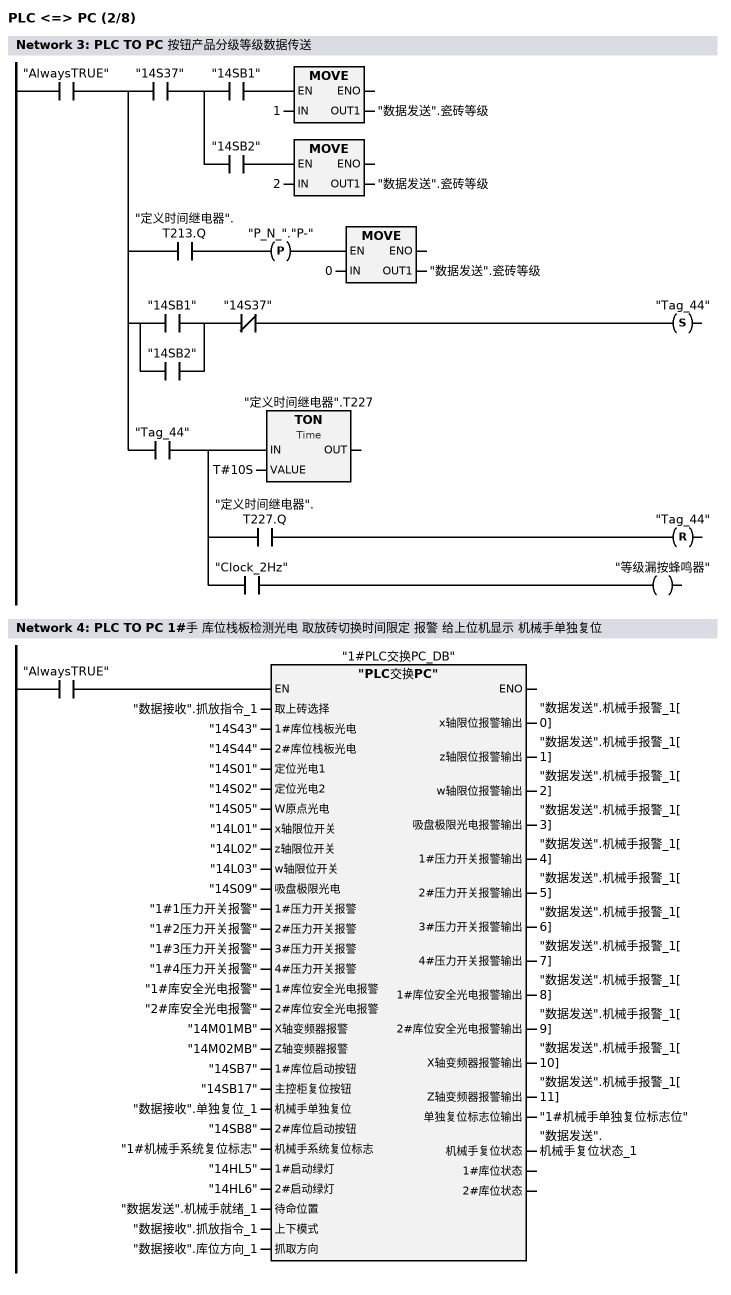
   #_w1 := "AlwaysTRUE" AND "14S37";
   IF #_w1 AND "14SB1" THEN "数据发送".瓷砖等级 := 1; END_IF;
   IF #_w1 AND "14SB2" THEN "数据发送".瓷砖等级 := 2; END_IF;
   #_w2 := "AlwaysTRUE" AND "定义时间继电器".T213.Q;
   #_w3 := #_w2 AND NOT "P_N_"."P-";   // rising edge
   "P_N_"."P-" := #_w2;
   IF #_w3 THEN "数据发送".瓷砖等级 := 0; END_IF;
   IF "AlwaysTRUE" AND ("14SB1" OR "14SB2") AND NOT "14S37" THEN "Tag_44" := TRUE; END_IF;
   #_w4 := "AlwaysTRUE" AND "Tag_44";
   "定义时间继电器".T227.TON(IN := #_w4, PT := T#10S);   // TON coil
   IF #_w4 AND "定义时间继电器".T227.Q THEN "Tag_44" := FALSE; END_IF;
   "等级漏按蜂鸣器" := #_w4 AND "Clock_2Hz";
END_REGION

REGION Network 4: PLC TO PC 1#手 库位栈板检测光电 取放砖切换时间限定 报警 给上位机显示 机械手单独复位
   RUNG wire#powerrail
      Contact( "AlwaysTRUE" )
      "1#PLC交换PC_DB"(取上砖选择 := "数据接收".抓放指令_1, "1#库位栈板光电" := "14S43", "2#库位栈板光电" := "14S44", 定位光电1 := "14S01", 定位光电2 := "14S02", W原点光电 := "14S05", x轴限位开关 := "14L01", z轴限位开关 := "14L02", w轴限位开关 := "14L03", 吸盘极限光电 := "14S09", "1#压力开关报警" := "1#1压力开关报警", "2#压力开关报警" := "1#2压力开关报警", "3#压力开关报警" := "1#3压力开关报警", "4#压力开关报警" := "1#4压力开关报警", "1#库位安全光电报警" := "1#库安全光电报警", "2#库位安全光电报警" := "2#库安全光电报警", X轴变频器报警 := "14M01MB", Z轴变频器报警 := "14M02MB", "1#库位启动按钮" := "14SB7", 主控柜复位按钮 := "14SB17", 机械手单独复位 := "数据接收".单独复位_1, "2#库位启动按钮" := "14SB8", 机械手系统复位标志 := "1#机械手系统复位标志", "1#启动绿灯" := "14HL5", "2#启动绿灯" := "14HL6", 待命位置 := "数据发送".机械手就绪_1, 上下模式 := "数据接收".抓放指令_1, 抓取方向 := "数据接收".库位方向_1, x轴限位报警输出 => "数据发送".机械手报警_1[0], z轴限位报警输出 => "数据发送".机械手报警_1[1], w轴限位报警输出 => "数据发送".机械手报警_1[2], 吸盘极限光电报警输出 => "数据发送".机械手报警_1[3], "1#压力开关报警输出" => "数据发送".机械手报警_1[4], "2#压力开关报警输出" => "数据发送".机械手报警_1[5], "3#压力开关报警输出" => "数据发送".机械手报警_1[6], "4#压力开关报警输出" => "数据发送".机械手报警_1[7], "1#库位安全光电报警输出" => "数据发送".机械手报警_1[8], "2#库位安全光电报警输出" => "数据发送".机械手报警_1[9], X轴变频器报警输出 => "数据发送".机械手报警_1[10], Z轴变频器报警输出 => "数据发送".机械手报警_1[11], 单独复位标志位输出 => "1#机械手单独复位标志位", 机械手复位状态 => "数据发送".机械手复位状态_1, "1#库位状态" =>, "2#库位状态" =>)
   END_RUNG
   // the same network as SCL:
   IF "AlwaysTRUE" THEN
       "1#PLC交换PC_DB"(取上砖选择 := "数据接收".抓放指令_1,   // "PLC交换PC"
                      "1#库位栈板光电" := "14S43",
                      "2#库位栈板光电" := "14S44",
                      定位光电1 := "14S01",
                      定位光电2 := "14S02",
                      W原点光电 := "14S05",
                      x轴限位开关 := "14L01",
                      z轴限位开关 := "14L02",
                      w轴限位开关 := "14L03",
                      吸盘极限光电 := "14S09",
                      "1#压力开关报警" := "1#1压力开关报警",
                      "2#压力开关报警" := "1#2压力开关报警",
                      "3#压力开关报警" := "1#3压力开关报警",
                      "4#压力开关报警" := "1#4压力开关报警",
                      "1#库位安全光电报警" := "1#库安全光电报警",
                      "2#库位安全光电报警" := "2#库安全光电报警",
                      X轴变频器报警 := "14M01MB",
                      Z轴变频器报警 := "14M02MB",
                      "1#库位启动按钮" := "14SB7",
                      主控柜复位按钮 := "14SB17",
                      机械手单独复位 := "数据接收".单独复位_1,
                      "2#库位启动按钮" := "14SB8",
                      机械手系统复位标志 := "1#机械手系统复位标志",
                      "1#启动绿灯" := "14HL5",
                      "2#启动绿灯" := "14HL6",
                      待命位置 := "数据发送".机械手就绪_1,
                      上下模式 := "数据接收".抓放指令_1,
                      抓取方向 := "数据接收".库位方向_1,
                      x轴限位报警输出 => "数据发送".机械手报警_1[0],
                      z轴限位报警输出 => "数据发送".机械手报警_1[1],
                      w轴限位报警输出 => "数据发送".机械手报警_1[2],
                      吸盘极限光电报警输出 => "数据发送".机械手报警_1[3],
                      "1#压力开关报警输出" => "数据发送".机械手报警_1[4],
                      "2#压力开关报警输出" => "数据发送".机械手报警_1[5],
                      "3#压力开关报警输出" => "数据发送".机械手报警_1[6],
                      "4#压力开关报警输出" => "数据发送".机械手报警_1[7],
                      "1#库位安全光电报警输出" => "数据发送".机械手报警_1[8],
                      "2#库位安全光电报警输出" => "数据发送".机械手报警_1[9],
                      X轴变频器报警输出 => "数据发送".机械手报警_1[10],
                      Z轴变频器报警输出 => "数据发送".机械手报警_1[11],
                      单独复位标志位输出 => "1#机械手单独复位标志位",
                      机械手复位状态 => "数据发送".机械手复位状态_1);
   END_IF;
END_REGION

REGION Network 5: PLC TO PC 2#手 库位栈板检测光电 取放砖切换时间限定 报警 给上位机显示 机械手单独复位
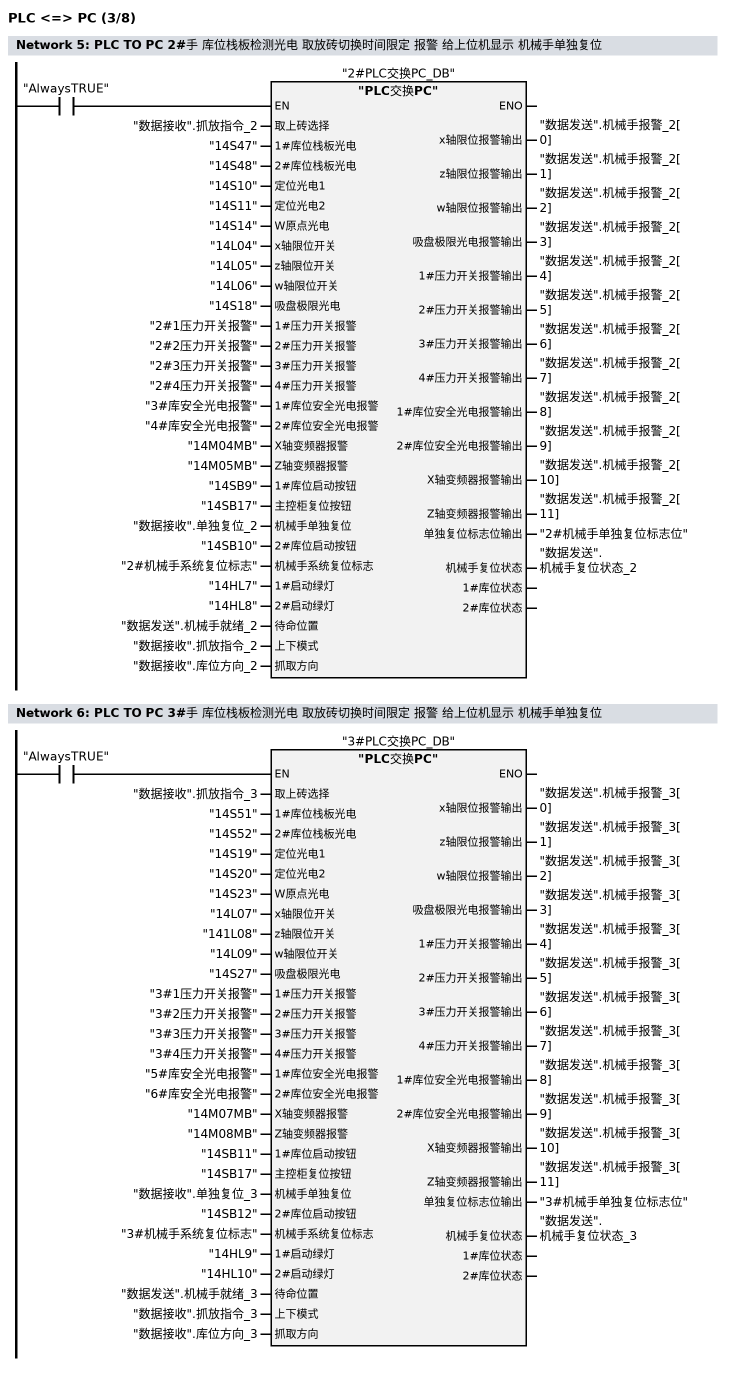
   RUNG wire#powerrail
      Contact( "AlwaysTRUE" )
      "2#PLC交换PC_DB"(取上砖选择 := "数据接收".抓放指令_2, "1#库位栈板光电" := "14S47", "2#库位栈板光电" := "14S48", 定位光电1 := "14S10", 定位光电2 := "14S11", W原点光电 := "14S14", x轴限位开关 := "14L04", z轴限位开关 := "14L05", w轴限位开关 := "14L06", 吸盘极限光电 := "14S18", "1#压力开关报警" := "2#1压力开关报警", "2#压力开关报警" := "2#2压力开关报警", "3#压力开关报警" := "2#3压力开关报警", "4#压力开关报警" := "2#4压力开关报警", "1#库位安全光电报警" := "3#库安全光电报警", "2#库位安全光电报警" := "4#库安全光电报警", X轴变频器报警 := "14M04MB", Z轴变频器报警 := "14M05MB", "1#库位启动按钮" := "14SB9", 主控柜复位按钮 := "14SB17", 机械手单独复位 := "数据接收".单独复位_2, "2#库位启动按钮" := "14SB10", 机械手系统复位标志 := "2#机械手系统复位标志", "1#启动绿灯" := "14HL7", "2#启动绿灯" := "14HL8", 待命位置 := "数据发送".机械手就绪_2, 上下模式 := "数据接收".抓放指令_2, 抓取方向 := "数据接收".库位方向_2, x轴限位报警输出 => "数据发送".机械手报警_2[0], z轴限位报警输出 => "数据发送".机械手报警_2[1], w轴限位报警输出 => "数据发送".机械手报警_2[2], 吸盘极限光电报警输出 => "数据发送".机械手报警_2[3], "1#压力开关报警输出" => "数据发送".机械手报警_2[4], "2#压力开关报警输出" => "数据发送".机械手报警_2[5], "3#压力开关报警输出" => "数据发送".机械手报警_2[6], "4#压力开关报警输出" => "数据发送".机械手报警_2[7], "1#库位安全光电报警输出" => "数据发送".机械手报警_2[8], "2#库位安全光电报警输出" => "数据发送".机械手报警_2[9], X轴变频器报警输出 => "数据发送".机械手报警_2[10], Z轴变频器报警输出 => "数据发送".机械手报警_2[11], 单独复位标志位输出 => "2#机械手单独复位标志位", 机械手复位状态 => "数据发送".机械手复位状态_2, "1#库位状态" =>, "2#库位状态" =>)
   END_RUNG
   // the same network as SCL:
   IF "AlwaysTRUE" THEN
       "2#PLC交换PC_DB"(取上砖选择 := "数据接收".抓放指令_2,   // "PLC交换PC"
                      "1#库位栈板光电" := "14S47",
                      "2#库位栈板光电" := "14S48",
                      定位光电1 := "14S10",
                      定位光电2 := "14S11",
                      W原点光电 := "14S14",
                      x轴限位开关 := "14L04",
                      z轴限位开关 := "14L05",
                      w轴限位开关 := "14L06",
                      吸盘极限光电 := "14S18",
                      "1#压力开关报警" := "2#1压力开关报警",
                      "2#压力开关报警" := "2#2压力开关报警",
                      "3#压力开关报警" := "2#3压力开关报警",
                      "4#压力开关报警" := "2#4压力开关报警",
                      "1#库位安全光电报警" := "3#库安全光电报警",
                      "2#库位安全光电报警" := "4#库安全光电报警",
                      X轴变频器报警 := "14M04MB",
                      Z轴变频器报警 := "14M05MB",
                      "1#库位启动按钮" := "14SB9",
                      主控柜复位按钮 := "14SB17",
                      机械手单独复位 := "数据接收".单独复位_2,
                      "2#库位启动按钮" := "14SB10",
                      机械手系统复位标志 := "2#机械手系统复位标志",
                      "1#启动绿灯" := "14HL7",
                      "2#启动绿灯" := "14HL8",
                      待命位置 := "数据发送".机械手就绪_2,
                      上下模式 := "数据接收".抓放指令_2,
                      抓取方向 := "数据接收".库位方向_2,
                      x轴限位报警输出 => "数据发送".机械手报警_2[0],
                      z轴限位报警输出 => "数据发送".机械手报警_2[1],
                      w轴限位报警输出 => "数据发送".机械手报警_2[2],
                      吸盘极限光电报警输出 => "数据发送".机械手报警_2[3],
                      "1#压力开关报警输出" => "数据发送".机械手报警_2[4],
                      "2#压力开关报警输出" => "数据发送".机械手报警_2[5],
                      "3#压力开关报警输出" => "数据发送".机械手报警_2[6],
                      "4#压力开关报警输出" => "数据发送".机械手报警_2[7],
                      "1#库位安全光电报警输出" => "数据发送".机械手报警_2[8],
                      "2#库位安全光电报警输出" => "数据发送".机械手报警_2[9],
                      X轴变频器报警输出 => "数据发送".机械手报警_2[10],
                      Z轴变频器报警输出 => "数据发送".机械手报警_2[11],
                      单独复位标志位输出 => "2#机械手单独复位标志位",
                      机械手复位状态 => "数据发送".机械手复位状态_2);
   END_IF;
END_REGION

REGION Network 6: PLC TO PC 3#手 库位栈板检测光电 取放砖切换时间限定 报警 给上位机显示 机械手单独复位
   RUNG wire#powerrail
      Contact( "AlwaysTRUE" )
      "3#PLC交换PC_DB"(取上砖选择 := "数据接收".抓放指令_3, "1#库位栈板光电" := "14S51", "2#库位栈板光电" := "14S52", 定位光电1 := "14S19", 定位光电2 := "14S20", W原点光电 := "14S23", x轴限位开关 := "14L07", z轴限位开关 := "141L08", w轴限位开关 := "14L09", 吸盘极限光电 := "14S27", "1#压力开关报警" := "3#1压力开关报警", "2#压力开关报警" := "3#2压力开关报警", "3#压力开关报警" := "3#3压力开关报警", "4#压力开关报警" := "3#4压力开关报警", "1#库位安全光电报警" := "5#库安全光电报警", "2#库位安全光电报警" := "6#库安全光电报警", X轴变频器报警 := "14M07MB", Z轴变频器报警 := "14M08MB", "1#库位启动按钮" := "14SB11", 主控柜复位按钮 := "14SB17", 机械手单独复位 := "数据接收".单独复位_3, "2#库位启动按钮" := "14SB12", 机械手系统复位标志 := "3#机械手系统复位标志", "1#启动绿灯" := "14HL9", "2#启动绿灯" := "14HL10", 待命位置 := "数据发送".机械手就绪_3, 上下模式 := "数据接收".抓放指令_3, 抓取方向 := "数据接收".库位方向_3, x轴限位报警输出 => "数据发送".机械手报警_3[0], z轴限位报警输出 => "数据发送".机械手报警_3[1], w轴限位报警输出 => "数据发送".机械手报警_3[2], 吸盘极限光电报警输出 => "数据发送".机械手报警_3[3], "1#压力开关报警输出" => "数据发送".机械手报警_3[4], "2#压力开关报警输出" => "数据发送".机械手报警_3[5], "3#压力开关报警输出" => "数据发送".机械手报警_3[6], "4#压力开关报警输出" => "数据发送".机械手报警_3[7], "1#库位安全光电报警输出" => "数据发送".机械手报警_3[8], "2#库位安全光电报警输出" => "数据发送".机械手报警_3[9], X轴变频器报警输出 => "数据发送".机械手报警_3[10], Z轴变频器报警输出 => "数据发送".机械手报警_3[11], 单独复位标志位输出 => "3#机械手单独复位标志位", 机械手复位状态 => "数据发送".机械手复位状态_3, "1#库位状态" =>, "2#库位状态" =>)
   END_RUNG
   // the same network as SCL:
   IF "AlwaysTRUE" THEN
       "3#PLC交换PC_DB"(取上砖选择 := "数据接收".抓放指令_3,   // "PLC交换PC"
                      "1#库位栈板光电" := "14S51",
                      "2#库位栈板光电" := "14S52",
                      定位光电1 := "14S19",
                      定位光电2 := "14S20",
                      W原点光电 := "14S23",
                      x轴限位开关 := "14L07",
                      z轴限位开关 := "141L08",
                      w轴限位开关 := "14L09",
                      吸盘极限光电 := "14S27",
                      "1#压力开关报警" := "3#1压力开关报警",
                      "2#压力开关报警" := "3#2压力开关报警",
                      "3#压力开关报警" := "3#3压力开关报警",
                      "4#压力开关报警" := "3#4压力开关报警",
                      "1#库位安全光电报警" := "5#库安全光电报警",
                      "2#库位安全光电报警" := "6#库安全光电报警",
                      X轴变频器报警 := "14M07MB",
                      Z轴变频器报警 := "14M08MB",
                      "1#库位启动按钮" := "14SB11",
                      主控柜复位按钮 := "14SB17",
                      机械手单独复位 := "数据接收".单独复位_3,
                      "2#库位启动按钮" := "14SB12",
                      机械手系统复位标志 := "3#机械手系统复位标志",
                      "1#启动绿灯" := "14HL9",
                      "2#启动绿灯" := "14HL10",
                      待命位置 := "数据发送".机械手就绪_3,
                      上下模式 := "数据接收".抓放指令_3,
                      抓取方向 := "数据接收".库位方向_3,
                      x轴限位报警输出 => "数据发送".机械手报警_3[0],
                      z轴限位报警输出 => "数据发送".机械手报警_3[1],
                      w轴限位报警输出 => "数据发送".机械手报警_3[2],
                      吸盘极限光电报警输出 => "数据发送".机械手报警_3[3],
                      "1#压力开关报警输出" => "数据发送".机械手报警_3[4],
                      "2#压力开关报警输出" => "数据发送".机械手报警_3[5],
                      "3#压力开关报警输出" => "数据发送".机械手报警_3[6],
                      "4#压力开关报警输出" => "数据发送".机械手报警_3[7],
                      "1#库位安全光电报警输出" => "数据发送".机械手报警_3[8],
                      "2#库位安全光电报警输出" => "数据发送".机械手报警_3[9],
                      X轴变频器报警输出 => "数据发送".机械手报警_3[10],
                      Z轴变频器报警输出 => "数据发送".机械手报警_3[11],
                      单独复位标志位输出 => "3#机械手单独复位标志位",
                      机械手复位状态 => "数据发送".机械手复位状态_3);
   END_IF;
END_REGION

REGION Network 7: PLC TO PC 4#手 库位栈板检测光电 取放砖切换时间限定 报警 给上位机显示 机械手单独复位
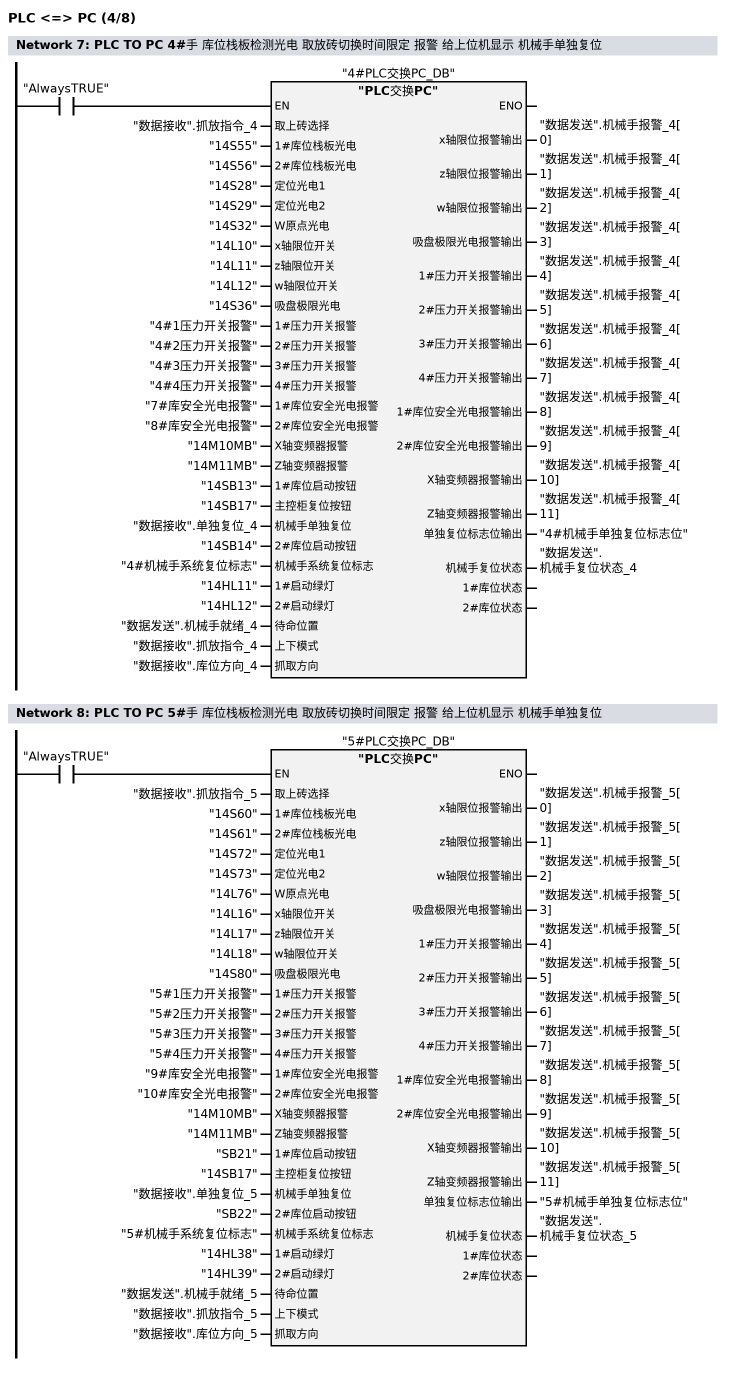
   RUNG wire#powerrail
      Contact( "AlwaysTRUE" )
      "4#PLC交换PC_DB"(取上砖选择 := "数据接收".抓放指令_4, "1#库位栈板光电" := "14S55", "2#库位栈板光电" := "14S56", 定位光电1 := "14S28", 定位光电2 := "14S29", W原点光电 := "14S32", x轴限位开关 := "14L10", z轴限位开关 := "14L11", w轴限位开关 := "14L12", 吸盘极限光电 := "14S36", "1#压力开关报警" := "4#1压力开关报警", "2#压力开关报警" := "4#2压力开关报警", "3#压力开关报警" := "4#3压力开关报警", "4#压力开关报警" := "4#4压力开关报警", "1#库位安全光电报警" := "7#库安全光电报警", "2#库位安全光电报警" := "8#库安全光电报警", X轴变频器报警 := "14M10MB", Z轴变频器报警 := "14M11MB", "1#库位启动按钮" := "14SB13", 主控柜复位按钮 := "14SB17", 机械手单独复位 := "数据接收".单独复位_4, "2#库位启动按钮" := "14SB14", 机械手系统复位标志 := "4#机械手系统复位标志", "1#启动绿灯" := "14HL11", "2#启动绿灯" := "14HL12", 待命位置 := "数据发送".机械手就绪_4, 上下模式 := "数据接收".抓放指令_4, 抓取方向 := "数据接收".库位方向_4, x轴限位报警输出 => "数据发送".机械手报警_4[0], z轴限位报警输出 => "数据发送".机械手报警_4[1], w轴限位报警输出 => "数据发送".机械手报警_4[2], 吸盘极限光电报警输出 => "数据发送".机械手报警_4[3], "1#压力开关报警输出" => "数据发送".机械手报警_4[4], "2#压力开关报警输出" => "数据发送".机械手报警_4[5], "3#压力开关报警输出" => "数据发送".机械手报警_4[6], "4#压力开关报警输出" => "数据发送".机械手报警_4[7], "1#库位安全光电报警输出" => "数据发送".机械手报警_4[8], "2#库位安全光电报警输出" => "数据发送".机械手报警_4[9], X轴变频器报警输出 => "数据发送".机械手报警_4[10], Z轴变频器报警输出 => "数据发送".机械手报警_4[11], 单独复位标志位输出 => "4#机械手单独复位标志位", 机械手复位状态 => "数据发送".机械手复位状态_4, "1#库位状态" =>, "2#库位状态" =>)
   END_RUNG
   // the same network as SCL:
   IF "AlwaysTRUE" THEN
       "4#PLC交换PC_DB"(取上砖选择 := "数据接收".抓放指令_4,   // "PLC交换PC"
                      "1#库位栈板光电" := "14S55",
                      "2#库位栈板光电" := "14S56",
                      定位光电1 := "14S28",
                      定位光电2 := "14S29",
                      W原点光电 := "14S32",
                      x轴限位开关 := "14L10",
                      z轴限位开关 := "14L11",
                      w轴限位开关 := "14L12",
                      吸盘极限光电 := "14S36",
                      "1#压力开关报警" := "4#1压力开关报警",
                      "2#压力开关报警" := "4#2压力开关报警",
                      "3#压力开关报警" := "4#3压力开关报警",
                      "4#压力开关报警" := "4#4压力开关报警",
                      "1#库位安全光电报警" := "7#库安全光电报警",
                      "2#库位安全光电报警" := "8#库安全光电报警",
                      X轴变频器报警 := "14M10MB",
                      Z轴变频器报警 := "14M11MB",
                      "1#库位启动按钮" := "14SB13",
                      主控柜复位按钮 := "14SB17",
                      机械手单独复位 := "数据接收".单独复位_4,
                      "2#库位启动按钮" := "14SB14",
                      机械手系统复位标志 := "4#机械手系统复位标志",
                      "1#启动绿灯" := "14HL11",
                      "2#启动绿灯" := "14HL12",
                      待命位置 := "数据发送".机械手就绪_4,
                      上下模式 := "数据接收".抓放指令_4,
                      抓取方向 := "数据接收".库位方向_4,
                      x轴限位报警输出 => "数据发送".机械手报警_4[0],
                      z轴限位报警输出 => "数据发送".机械手报警_4[1],
                      w轴限位报警输出 => "数据发送".机械手报警_4[2],
                      吸盘极限光电报警输出 => "数据发送".机械手报警_4[3],
                      "1#压力开关报警输出" => "数据发送".机械手报警_4[4],
                      "2#压力开关报警输出" => "数据发送".机械手报警_4[5],
                      "3#压力开关报警输出" => "数据发送".机械手报警_4[6],
                      "4#压力开关报警输出" => "数据发送".机械手报警_4[7],
                      "1#库位安全光电报警输出" => "数据发送".机械手报警_4[8],
                      "2#库位安全光电报警输出" => "数据发送".机械手报警_4[9],
                      X轴变频器报警输出 => "数据发送".机械手报警_4[10],
                      Z轴变频器报警输出 => "数据发送".机械手报警_4[11],
                      单独复位标志位输出 => "4#机械手单独复位标志位",
                      机械手复位状态 => "数据发送".机械手复位状态_4);
   END_IF;
END_REGION

REGION Network 8: PLC TO PC 5#手 库位栈板检测光电 取放砖切换时间限定 报警 给上位机显示 机械手单独复位
   RUNG wire#powerrail
      Contact( "AlwaysTRUE" )
      "5#PLC交换PC_DB"(取上砖选择 := "数据接收".抓放指令_5, "1#库位栈板光电" := "14S60", "2#库位栈板光电" := "14S61", 定位光电1 := "14S72", 定位光电2 := "14S73", W原点光电 := "14L76", x轴限位开关 := "14L16", z轴限位开关 := "14L17", w轴限位开关 := "14L18", 吸盘极限光电 := "14S80", "1#压力开关报警" := "5#1压力开关报警", "2#压力开关报警" := "5#2压力开关报警", "3#压力开关报警" := "5#3压力开关报警", "4#压力开关报警" := "5#4压力开关报警", "1#库位安全光电报警" := "9#库安全光电报警", "2#库位安全光电报警" := "10#库安全光电报警", X轴变频器报警 := "14M10MB", Z轴变频器报警 := "14M11MB", "1#库位启动按钮" := "SB21", 主控柜复位按钮 := "14SB17", 机械手单独复位 := "数据接收".单独复位_5, "2#库位启动按钮" := "SB22", 机械手系统复位标志 := "5#机械手系统复位标志", "1#启动绿灯" := "14HL38", "2#启动绿灯" := "14HL39", 待命位置 := "数据发送".机械手就绪_5, 上下模式 := "数据接收".抓放指令_5, 抓取方向 := "数据接收".库位方向_5, x轴限位报警输出 => "数据发送".机械手报警_5[0], z轴限位报警输出 => "数据发送".机械手报警_5[1], w轴限位报警输出 => "数据发送".机械手报警_5[2], 吸盘极限光电报警输出 => "数据发送".机械手报警_5[3], "1#压力开关报警输出" => "数据发送".机械手报警_5[4], "2#压力开关报警输出" => "数据发送".机械手报警_5[5], "3#压力开关报警输出" => "数据发送".机械手报警_5[6], "4#压力开关报警输出" => "数据发送".机械手报警_5[7], "1#库位安全光电报警输出" => "数据发送".机械手报警_5[8], "2#库位安全光电报警输出" => "数据发送".机械手报警_5[9], X轴变频器报警输出 => "数据发送".机械手报警_5[10], Z轴变频器报警输出 => "数据发送".机械手报警_5[11], 单独复位标志位输出 => "5#机械手单独复位标志位", 机械手复位状态 => "数据发送".机械手复位状态_5, "1#库位状态" =>, "2#库位状态" =>)
   END_RUNG
   // the same network as SCL:
   IF "AlwaysTRUE" THEN
       "5#PLC交换PC_DB"(取上砖选择 := "数据接收".抓放指令_5,   // "PLC交换PC"
                      "1#库位栈板光电" := "14S60",
                      "2#库位栈板光电" := "14S61",
                      定位光电1 := "14S72",
                      定位光电2 := "14S73",
                      W原点光电 := "14L76",
                      x轴限位开关 := "14L16",
                      z轴限位开关 := "14L17",
                      w轴限位开关 := "14L18",
                      吸盘极限光电 := "14S80",
                      "1#压力开关报警" := "5#1压力开关报警",
                      "2#压力开关报警" := "5#2压力开关报警",
                      "3#压力开关报警" := "5#3压力开关报警",
                      "4#压力开关报警" := "5#4压力开关报警",
                      "1#库位安全光电报警" := "9#库安全光电报警",
                      "2#库位安全光电报警" := "10#库安全光电报警",
                      X轴变频器报警 := "14M10MB",
                      Z轴变频器报警 := "14M11MB",
                      "1#库位启动按钮" := "SB21",
                      主控柜复位按钮 := "14SB17",
                      机械手单独复位 := "数据接收".单独复位_5,
                      "2#库位启动按钮" := "SB22",
                      机械手系统复位标志 := "5#机械手系统复位标志",
                      "1#启动绿灯" := "14HL38",
                      "2#启动绿灯" := "14HL39",
                      待命位置 := "数据发送".机械手就绪_5,
                      上下模式 := "数据接收".抓放指令_5,
                      抓取方向 := "数据接收".库位方向_5,
                      x轴限位报警输出 => "数据发送".机械手报警_5[0],
                      z轴限位报警输出 => "数据发送".机械手报警_5[1],
                      w轴限位报警输出 => "数据发送".机械手报警_5[2],
                      吸盘极限光电报警输出 => "数据发送".机械手报警_5[3],
                      "1#压力开关报警输出" => "数据发送".机械手报警_5[4],
                      "2#压力开关报警输出" => "数据发送".机械手报警_5[5],
                      "3#压力开关报警输出" => "数据发送".机械手报警_5[6],
                      "4#压力开关报警输出" => "数据发送".机械手报警_5[7],
                      "1#库位安全光电报警输出" => "数据发送".机械手报警_5[8],
                      "2#库位安全光电报警输出" => "数据发送".机械手报警_5[9],
                      X轴变频器报警输出 => "数据发送".机械手报警_5[10],
                      Z轴变频器报警输出 => "数据发送".机械手报警_5[11],
                      单独复位标志位输出 => "5#机械手单独复位标志位",
                      机械手复位状态 => "数据发送".机械手复位状态_5);
   END_IF;
END_REGION

REGION Network 9: PLC TO PC 队列光电4
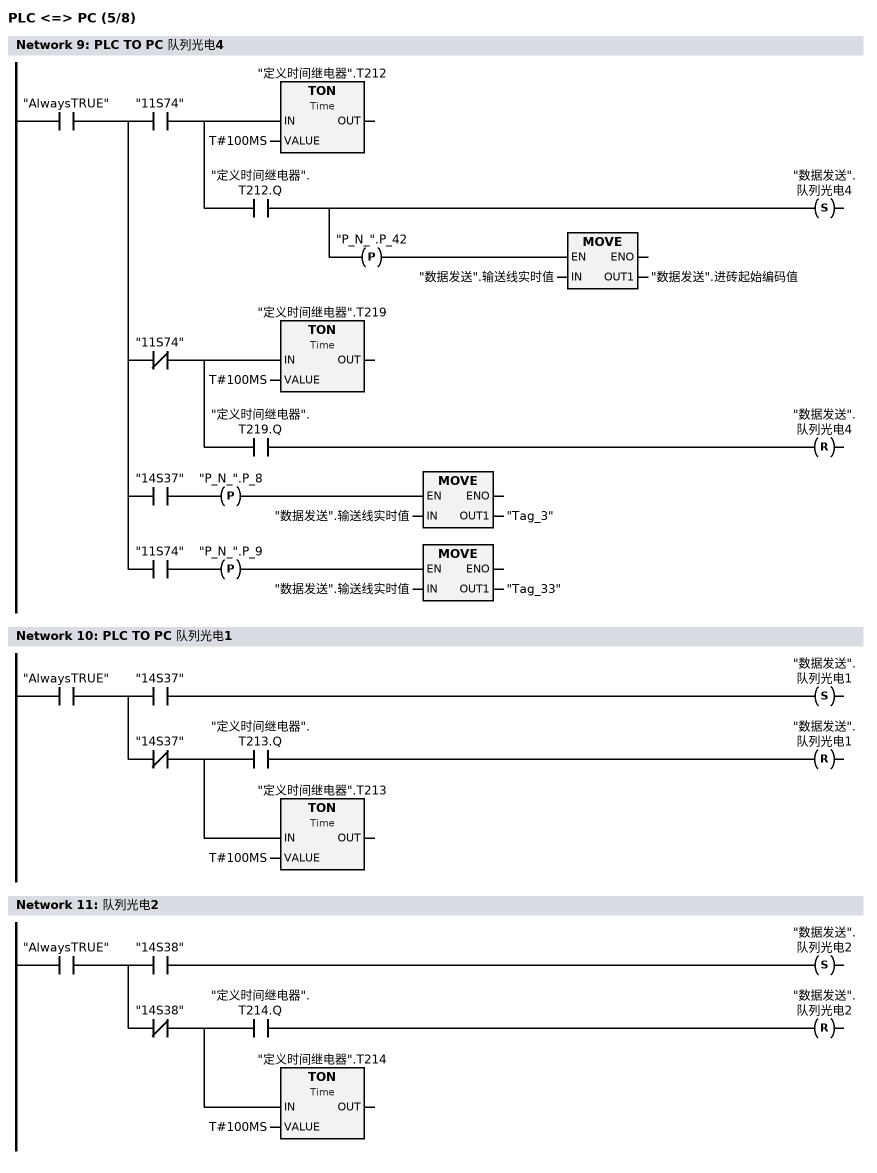
   #_w1 := "AlwaysTRUE" AND "11S74";
   "定义时间继电器".T212.TON(IN := #_w1, PT := T#100MS);   // TON coil
   #_w2 := #_w1 AND "定义时间继电器".T212.Q;
   IF #_w2 THEN "数据发送".队列光电4 := TRUE; END_IF;
   #_w3 := #_w2 AND NOT "P_N_".P_42;   // rising edge
   "P_N_".P_42 := #_w2;
   IF #_w3 THEN "数据发送".进砖起始编码值 := "数据发送".输送线实时值; END_IF;
   #_w4 := "AlwaysTRUE" AND NOT "11S74";
   "定义时间继电器".T219.TON(IN := #_w4, PT := T#100MS);   // TON coil
   IF #_w4 AND "定义时间继电器".T219.Q THEN "数据发送".队列光电4 := FALSE; END_IF;
   #_w5 := "AlwaysTRUE" AND "14S37";
   #_w6 := #_w5 AND NOT "P_N_".P_8;   // rising edge
   "P_N_".P_8 := #_w5;
   IF #_w6 THEN "Tag_3" := "数据发送".输送线实时值; END_IF;
   #_w7 := "AlwaysTRUE" AND "11S74";
   #_w8 := #_w7 AND NOT "P_N_".P_9;   // rising edge
   "P_N_".P_9 := #_w7;
   IF #_w8 THEN "Tag_33" := "数据发送".输送线实时值; END_IF;
END_REGION

REGION Network 10: PLC TO PC 队列光电1
   IF "AlwaysTRUE" AND "14S37" THEN "数据发送".队列光电1 := TRUE; END_IF;
   #_w1 := "AlwaysTRUE" AND NOT "14S37";
   IF #_w1 AND "定义时间继电器".T213.Q THEN "数据发送".队列光电1 := FALSE; END_IF;
   "定义时间继电器".T213.TON(IN := #_w1, PT := T#100MS);   // TON coil
END_REGION

REGION Network 11: 队列光电2
   IF "AlwaysTRUE" AND "14S38" THEN "数据发送".队列光电2 := TRUE; END_IF;
   #_w1 := "AlwaysTRUE" AND NOT "14S38";
   IF #_w1 AND "定义时间继电器".T214.Q THEN "数据发送".队列光电2 := FALSE; END_IF;
   "定义时间继电器".T214.TON(IN := #_w1, PT := T#100MS);   // TON coil
END_REGION

REGION Network 12: 队列光电3
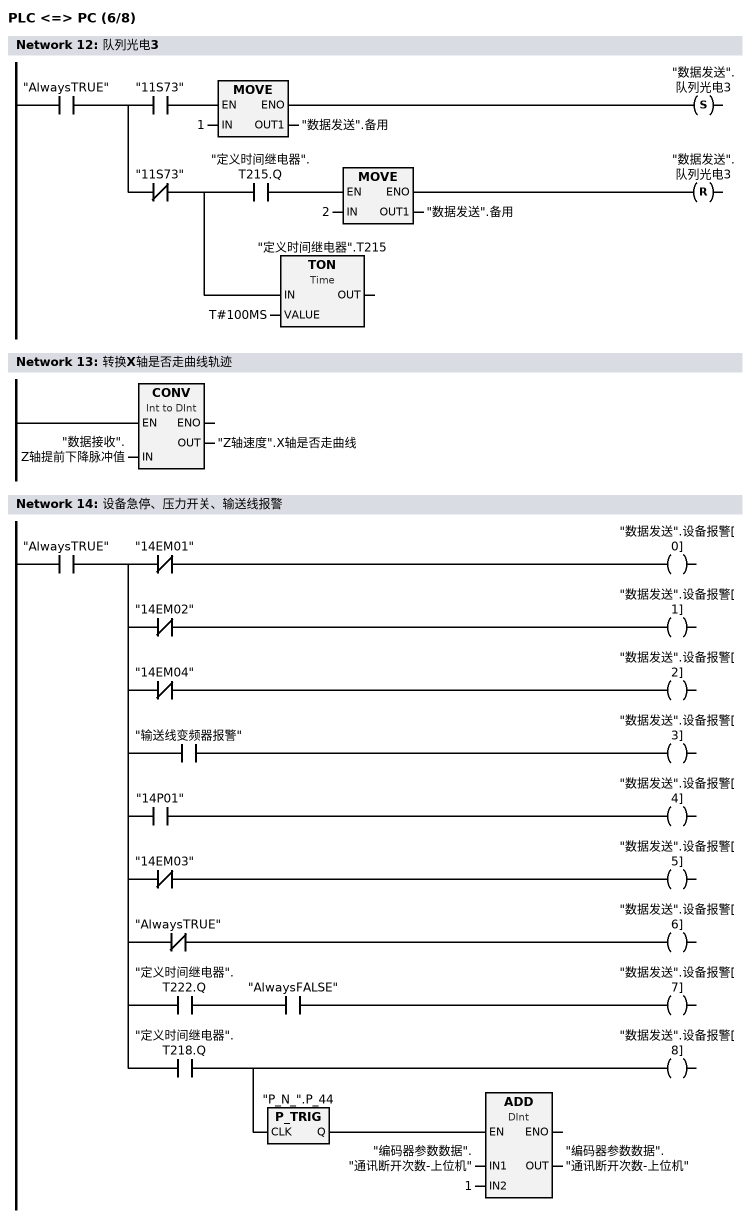
   IF "AlwaysTRUE" AND "11S73" THEN
       "数据发送".备用 := 1;
       "数据发送".队列光电3 := TRUE;
   END_IF;
   #_w1 := "AlwaysTRUE" AND NOT "11S73";
   IF #_w1 AND "定义时间继电器".T215.Q THEN
       "数据发送".备用 := 2;
       "数据发送".队列光电3 := FALSE;
   END_IF;
   "定义时间继电器".T215.TON(IN := #_w1, PT := T#100MS);   // TON coil
END_REGION

REGION Network 13: 转换X轴是否走曲线轨迹
   RUNG wire#powerrail
      { S7_Templates := "[SrcType := Int, DestType := DInt]" } Convert(in := "数据接收".Z轴提前下降脉冲值, out => "Z轴速度".X轴是否走曲线)
   END_RUNG
   // the same network as SCL:
   "Z轴速度".X轴是否走曲线 := INT_TO_DINT("数据接收".Z轴提前下降脉冲值);
END_REGION

REGION Network 14: 设备急停、压力开关、输送线报警
   RUNG wire#powerrail
      Contact( "AlwaysTRUE" )
      wire#w1
      I_Contact( "14EM01" )
      Coil( "数据发送".设备报警[0] )
   END_RUNG
   RUNG wire#w1
      I_Contact( "14EM02" )
      Coil( "数据发送".设备报警[1] )
   END_RUNG
   RUNG wire#w1
      I_Contact( "14EM04" )
      Coil( "数据发送".设备报警[2] )
   END_RUNG
   RUNG wire#w1
      Contact( "输送线变频器报警" )
      Coil( "数据发送".设备报警[3] )
   END_RUNG
   RUNG wire#w1
      Contact( "14P01" )
      Coil( "数据发送".设备报警[4] )
   END_RUNG
   RUNG wire#w1
      I_Contact( "14EM03" )
      Coil( "数据发送".设备报警[5] )
   END_RUNG
   RUNG wire#w1
      I_Contact( "AlwaysTRUE" )
      Coil( "数据发送".设备报警[6] )
   END_RUNG
   RUNG wire#w1
      Contact( "定义时间继电器".T222.Q )
      Contact( "AlwaysFALSE" )
      Coil( "数据发送".设备报警[7] )
   END_RUNG
   RUNG wire#w1
      Contact( "定义时间继电器".T218.Q )
      wire#w2
      Coil( "数据发送".设备报警[8] )
   END_RUNG
   RUNG wire#w2
      P_Trig( "P_N_".P_44 )
      { S7_Templates := "SrcType := DInt" } Add(in1 := "编码器参数数据"."通讯断开次数-上位机", in2 := 1, out => "编码器参数数据"."通讯断开次数-上位机")
   END_RUNG
   // the same network as SCL:
   "数据发送".设备报警[0] := "AlwaysTRUE" AND NOT "14EM01";
   "数据发送".设备报警[1] := "AlwaysTRUE" AND NOT "14EM02";
   "数据发送".设备报警[2] := "AlwaysTRUE" AND NOT "14EM04";
   "数据发送".设备报警[3] := "AlwaysTRUE" AND "输送线变频器报警";
   "数据发送".设备报警[4] := "AlwaysTRUE" AND "14P01";
   "数据发送".设备报警[5] := "AlwaysTRUE" AND NOT "14EM03";
   "数据发送".设备报警[6] := "AlwaysTRUE" AND NOT "AlwaysTRUE";
   "数据发送".设备报警[7] := "AlwaysTRUE" AND "定义时间继电器".T222.Q AND "AlwaysFALSE";
   "数据发送".设备报警[8] := "AlwaysTRUE" AND "定义时间继电器".T218.Q;
   #_w1 := "AlwaysTRUE" AND "定义时间继电器".T218.Q;
   #_w2 := #_w1 AND NOT "P_N_".P_44;   // rising edge
   "P_N_".P_44 := #_w1;
   IF #_w2 THEN "编码器参数数据"."通讯断开次数-上位机" := "编码器参数数据"."通讯断开次数-上位机" + 1; END_IF;
END_REGION

REGION Network 15: 换花色旋钮=>给上位机
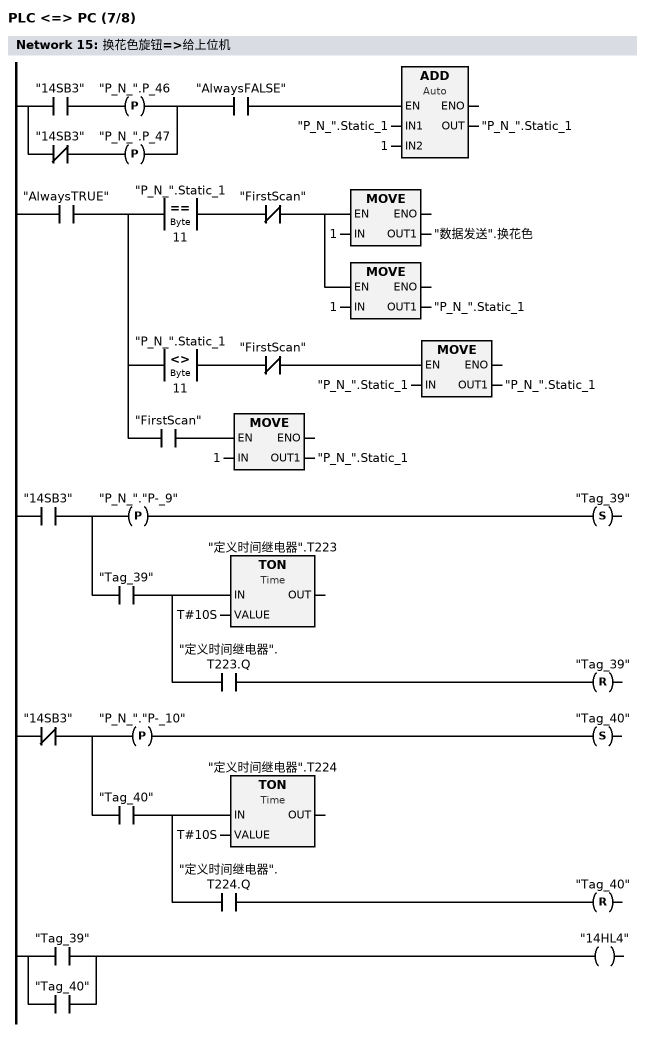
   #_w1 := "14SB3" AND NOT "P_N_".P_46;   // rising edge
   "P_N_".P_46 := "14SB3";
   #_w2 := NOT "14SB3" AND NOT "P_N_".P_47;   // rising edge
   "P_N_".P_47 := NOT "14SB3";
   IF (#_w1 OR #_w2) AND "AlwaysFALSE" THEN "P_N_".Static_1 := "P_N_".Static_1 + 1; END_IF;
   IF "AlwaysTRUE" AND ("P_N_".Static_1 = 11) AND NOT "FirstScan" THEN
       "数据发送".换花色 := 1;
       "P_N_".Static_1 := 1;
   END_IF;
   IF "AlwaysTRUE" AND ("P_N_".Static_1 <> 11) AND NOT "FirstScan" THEN
       "P_N_".Static_1 := "P_N_".Static_1;
   END_IF;
   IF "AlwaysTRUE" AND "FirstScan" THEN "P_N_".Static_1 := 1; END_IF;
   #_w3 := "14SB3" AND NOT "P_N_"."P-_9";   // rising edge
   "P_N_"."P-_9" := "14SB3";
   IF #_w3 THEN "Tag_39" := TRUE; END_IF;
   #_w4 := "14SB3" AND "Tag_39";
   "定义时间继电器".T223.TON(IN := #_w4, PT := T#10S);   // TON coil
   IF #_w4 AND "定义时间继电器".T223.Q THEN "Tag_39" := FALSE; END_IF;
   #_w5 := NOT "14SB3" AND NOT "P_N_"."P-_10";   // rising edge
   "P_N_"."P-_10" := NOT "14SB3";
   IF #_w5 THEN "Tag_40" := TRUE; END_IF;
   #_w6 := NOT "14SB3" AND "Tag_40";
   "定义时间继电器".T224.TON(IN := #_w6, PT := T#10S);   // TON coil
   IF #_w6 AND "定义时间继电器".T224.Q THEN "Tag_40" := FALSE; END_IF;
   "14HL4" := "Tag_39" OR "Tag_40";
END_REGION

REGION Network 16: 上位机询问是否可以砖放行 16询问结果传输
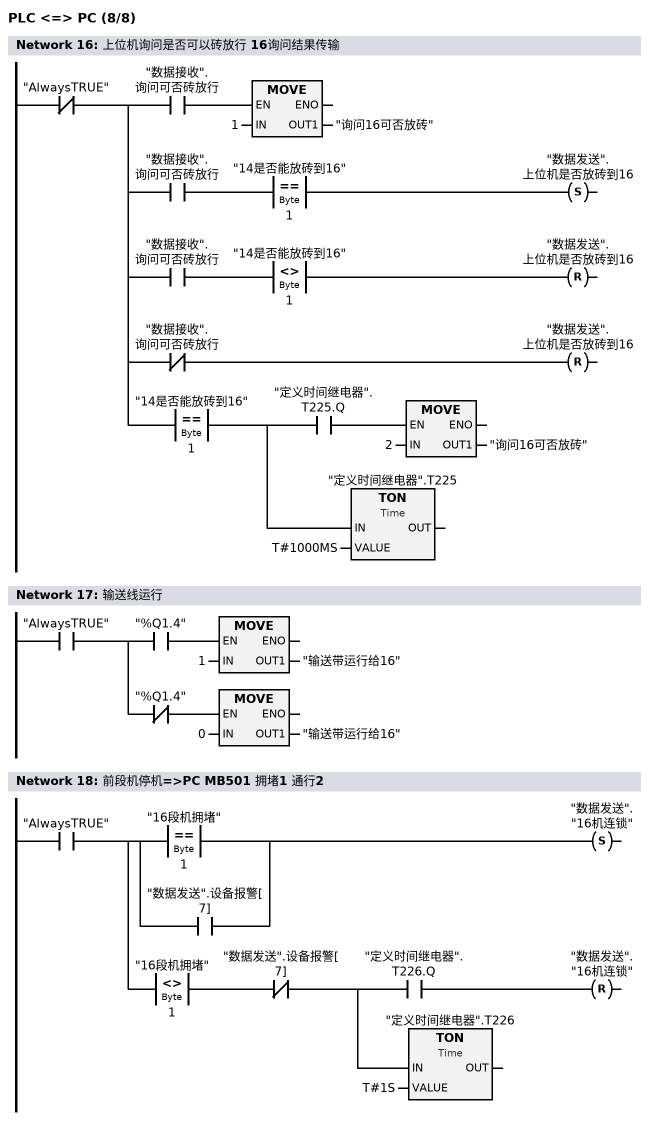
   IF NOT "AlwaysTRUE" AND "数据接收".询问可否砖放行 THEN "询问16可否放砖" := 1; END_IF;
   IF NOT "AlwaysTRUE" AND "数据接收".询问可否砖放行 AND ("14是否能放砖到16" = 1) THEN "数据发送".上位机是否放砖到16 := TRUE; END_IF;
   IF NOT "AlwaysTRUE" AND "数据接收".询问可否砖放行 AND ("14是否能放砖到16" <> 1) THEN "数据发送".上位机是否放砖到16 := FALSE; END_IF;
   IF NOT "AlwaysTRUE" AND NOT "数据接收".询问可否砖放行 THEN "数据发送".上位机是否放砖到16 := FALSE; END_IF;
   #_w1 := NOT "AlwaysTRUE" AND ("14是否能放砖到16" = 1);
   IF #_w1 AND "定义时间继电器".T225.Q THEN "询问16可否放砖" := 2; END_IF;
   "定义时间继电器".T225.TON(IN := #_w1, PT := T#1000MS);   // TON coil
END_REGION

REGION Network 17: 输送线运行
   RUNG wire#powerrail
      Contact( "AlwaysTRUE" )
      wire#w1
      Contact( "%Q1.4" )
      Move(in := 1, out1 => "输送带运行给16")
   END_RUNG
   RUNG wire#w1
      I_Contact( "%Q1.4" )
      Move(in := 0, out1 => "输送带运行给16")
   END_RUNG
   // the same network as SCL:
   IF "AlwaysTRUE" AND "%Q1.4" THEN "输送带运行给16" := 1; END_IF;
   IF "AlwaysTRUE" AND NOT "%Q1.4" THEN "输送带运行给16" := 0; END_IF;
END_REGION

REGION Network 18: 前段机停机=>PC MB501 拥堵1 通行2
   IF "AlwaysTRUE" AND (("16段机拥堵" = 1) OR "数据发送".设备报警[7]) THEN "数据发送"."16机连锁" := TRUE; END_IF;
   #_w1 := "AlwaysTRUE" AND ("16段机拥堵" <> 1) AND NOT "数据发送".设备报警[7];
   IF #_w1 AND "定义时间继电器".T226.Q THEN "数据发送"."16机连锁" := FALSE; END_IF;
   "定义时间继电器".T226.TON(IN := #_w1, PT := T#1S);   // TON coil
END_REGION
END_FUNCTION

// folder: 通讯/射频通信/射频通信

FUNCTION_BLOCK "F2射频读取切换功能块"   // FB15, LAD
{ S7_Optimized_Access := 'FALSE' }
VERSION : 0.1
   VAR_INPUT
      中断连接 : Bool;
      配置发送完成 : Bool;
      判断次数 : SInt;
      IO状态1 : Array[0..15] of Bool;
      IO状态2 : Array[0..15] of Bool;
      IO状态3 : Array[0..15] of Bool;
      IO状态4 : Array[0..15] of Bool;
      IO数据_1 : Array[0..5] of Byte;
      IO数据_2 : Array[0..5] of Byte;
      IO数据_3 : Array[0..5] of Byte;
      IO数据_4 : Array[0..5] of Byte;
   END_VAR
   VAR_IN_OUT
      清除指令 : Bool;
      读数据指令 : Bool;
      读UID指令 : Bool;
      IOSys : Byte;
      IO输出值_1 : Array[0..5] of Byte;
      IO输出值_2 : Array[0..5] of Byte;
      IO输出值_3 : Array[0..5] of Byte;
      IO输出值_4 : Array[0..5] of Byte;
      栈板有无_1 : Byte;
      栈板有无_2 : Byte;
      栈板有无_3 : Byte;
      栈板有无_4 : Byte;
   END_VAR
   VAR
      配置完成延时 : Bool;
      读数据状态 : Bool;
      配置完成定时器 : IEC_TIMER;
      清除指令定时器 : IEC_TIMER;
      读数据定时器 : IEC_TIMER;
      读UID定时器 : IEC_TIMER;
      判断定时器_1 : IEC_TIMER;
      判断定时器_2 : IEC_TIMER;
      判断定时器_3 : IEC_TIMER;
      判断定时器_4 : IEC_TIMER;
      读取过滤定时器_5 : IEC_TIMER;
      读取过滤定时器_6 : IEC_TIMER;
      读取过滤定时器_7 : IEC_TIMER;
      读取过滤定时器_8 : IEC_TIMER;
      IO输出中间值_1 : Array[0..5] of Byte;
      IO输出中间值_2 : Array[0..5] of Byte;
      IO输出中间值_3 : Array[0..5] of Byte;
      IO输出中间值_4 : Array[0..5] of Byte;
      栈板状态_1 : Byte;   // 1有2无
      栈板状态_2 : Byte;
      栈板状态_3 : Byte;
      栈板状态_4 : Byte;
      栈板中间状态_1 : Byte;   // 1有2无
      栈板中间状态_2 : Byte;
      栈板中间状态_3 : Byte;
      栈板中间状态_4 : Byte;
      次数1 : SInt;
      次数2 : SInt;
      次数3 : SInt;
      次数4 : SInt;
      读取P1 : Bool;
      读取P2 : Bool;
      读取P3 : Bool;
      读取P4 : Bool;
      IO成功_1 : Bool;
      IO成功_2 : Bool;
      IO成功_3 : Bool;
      IO成功_4 : Bool;
      读取完成 : Bool;
      UID状态值_1 : Bool;
      UID状态值_2 : Bool;
      UID状态值_3 : Bool;
      UID状态值_4 : Bool;
      读取P : Bool;
      IO故障_1 : Bool;
      IO故障_2 : Bool;
      IO故障_3 : Bool;
      IO故障_4 : Bool;
   END_VAR
   VAR_TEMP   // added for the SCL form of the ladder/FBD networks
      _w1 : Bool;
      _w2 : Bool;
      _w3 : Bool;
      _w4 : Bool;
      _w5 : Bool;
      _w6 : Bool;
      _w7 : Bool;
      _w8 : Bool;
      _w9 : Bool;
      _w10 : Bool;
      _w11 : Bool;
      _w12 : Bool;
      _w13 : Bool;
      _w14 : Bool;
      _w15 : Bool;
      _w16 : Bool;
   END_VAR
BEGIN

REGION Network 1
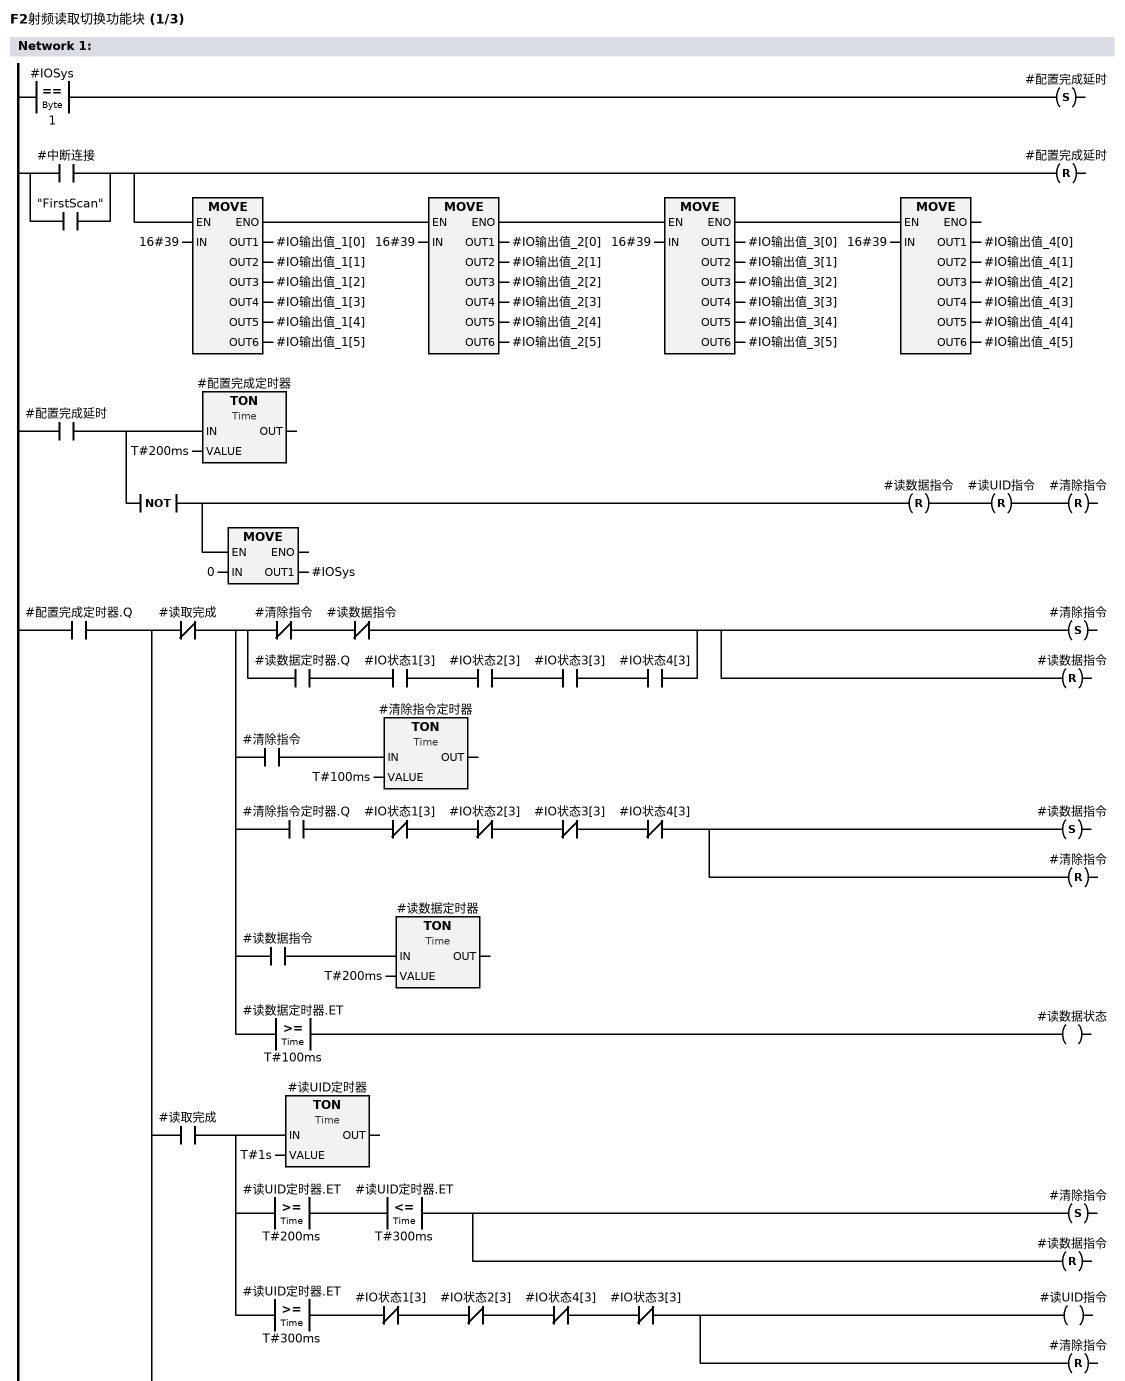
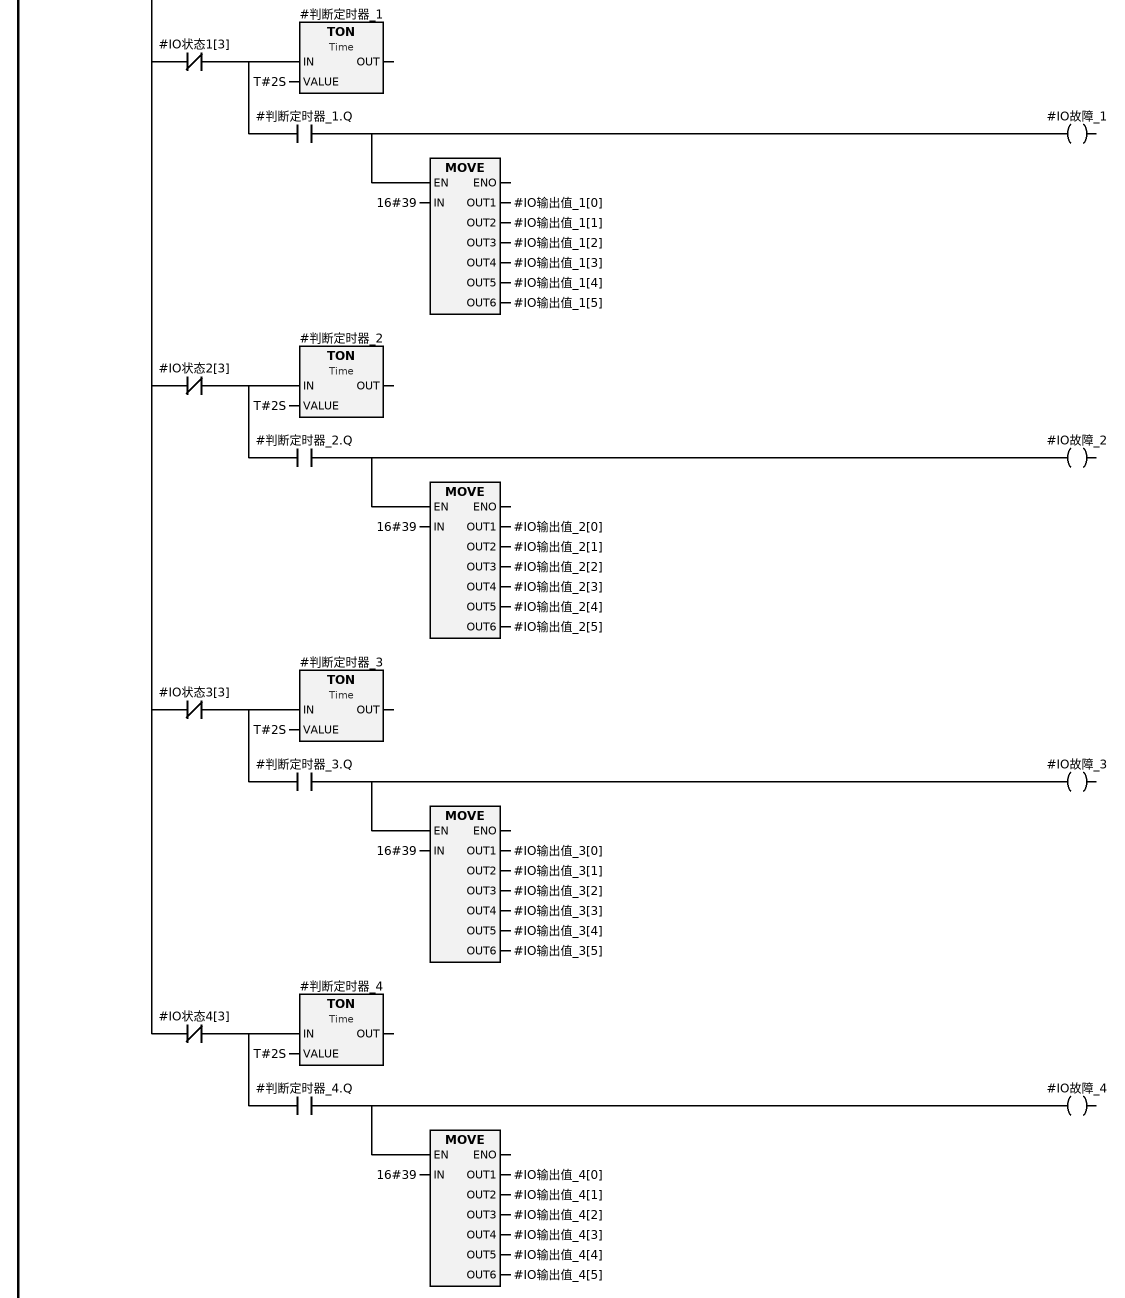
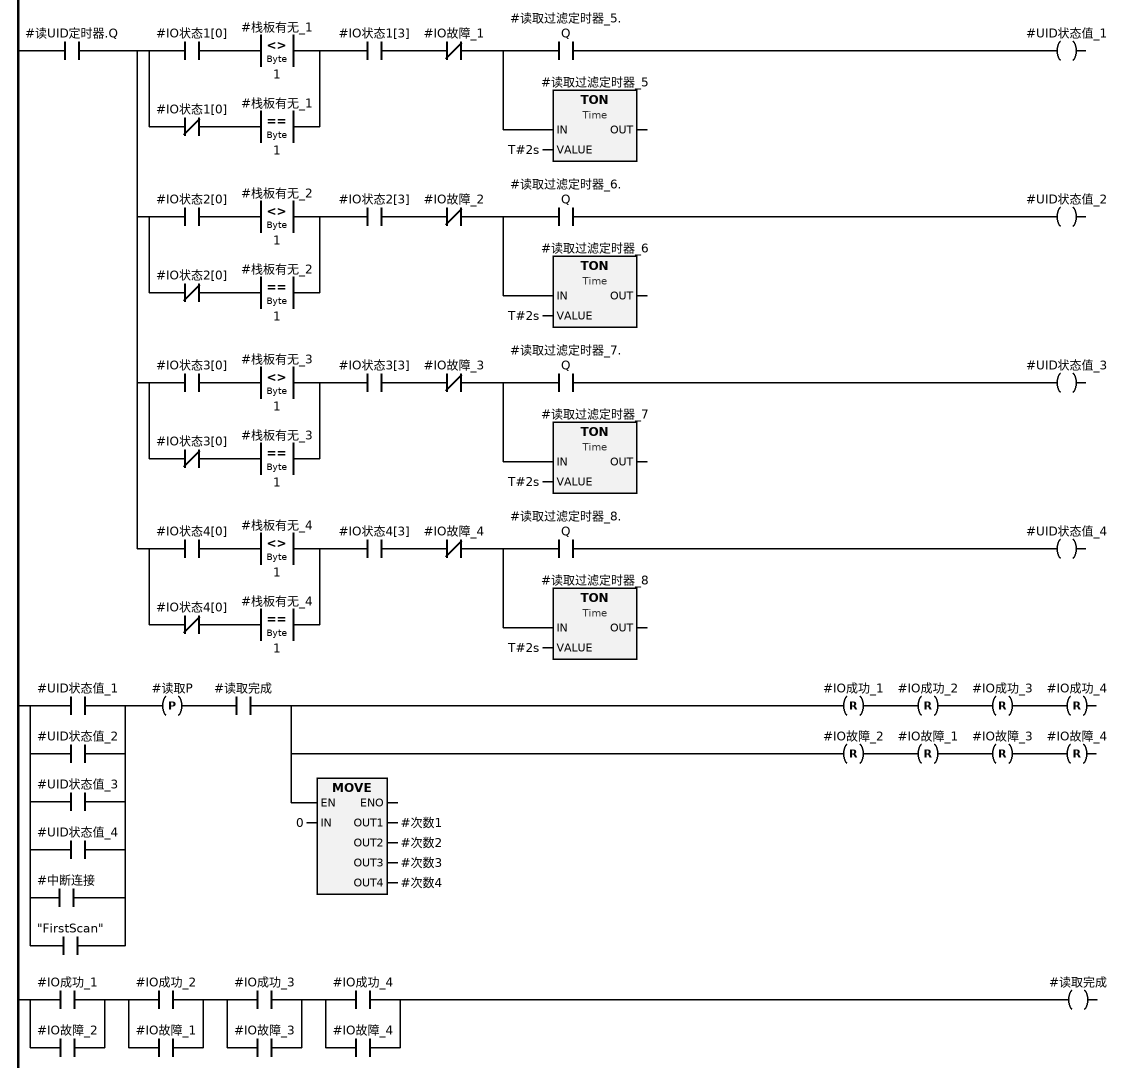
   IF #IOSys = 1 THEN #配置完成延时 := TRUE; END_IF;
   IF #中断连接 OR "FirstScan" THEN
       #配置完成延时 := FALSE;
       #IO输出值_1[0] := 16#39;
       #IO输出值_1[1] := 16#39;
       #IO输出值_1[2] := 16#39;
       #IO输出值_1[3] := 16#39;
       #IO输出值_1[4] := 16#39;
       #IO输出值_1[5] := 16#39;
       #IO输出值_2[0] := 16#39;
       #IO输出值_2[1] := 16#39;
       #IO输出值_2[2] := 16#39;
       #IO输出值_2[3] := 16#39;
       #IO输出值_2[4] := 16#39;
       #IO输出值_2[5] := 16#39;
       #IO输出值_3[0] := 16#39;
       #IO输出值_3[1] := 16#39;
       #IO输出值_3[2] := 16#39;
       #IO输出值_3[3] := 16#39;
       #IO输出值_3[4] := 16#39;
       #IO输出值_3[5] := 16#39;
       #IO输出值_4[0] := 16#39;
       #IO输出值_4[1] := 16#39;
       #IO输出值_4[2] := 16#39;
       #IO输出值_4[3] := 16#39;
       #IO输出值_4[4] := 16#39;
       #IO输出值_4[5] := 16#39;
   END_IF;
   #配置完成定时器.TON(IN := #配置完成延时, PT := T#200ms);   // TON coil
   IF NOT #配置完成延时 THEN
       #读数据指令 := FALSE;
       #读UID指令 := FALSE;
       #清除指令 := FALSE;
       #IOSys := 0;
   END_IF;
   #_w1 := #配置完成定时器.Q AND NOT #读取完成;
   #_w2 := #_w1 AND ((NOT #清除指令 AND NOT #读数据指令) OR (#读数据定时器.Q AND #IO状态1[3] AND #IO状态2[3] AND #IO状态3[3] AND #IO状态4[3]));
   IF #_w2 THEN
       #清除指令 := TRUE;
       #读数据指令 := FALSE;
   END_IF;
   #清除指令定时器.TON(IN := #_w1 AND #清除指令, PT := T#100ms);   // TON coil
   IF #_w1 AND #清除指令定时器.Q AND NOT #IO状态1[3] AND NOT #IO状态2[3] AND NOT #IO状态3[3] AND NOT #IO状态4[3] THEN
       #读数据指令 := TRUE;
       #清除指令 := FALSE;
   END_IF;
   #读数据定时器.TON(IN := #_w1 AND #读数据指令, PT := T#200ms);   // TON coil
   #读数据状态 := #_w1 AND (#读数据定时器.ET >= T#100ms);
   #_w3 := #配置完成定时器.Q AND #读取完成;
   #读UID定时器.TON(IN := #_w3, PT := T#1s);   // TON coil
   IF #_w3 AND (#读UID定时器.ET >= T#200ms) AND (#读UID定时器.ET <= T#300ms) THEN
       #清除指令 := TRUE;
       #读数据指令 := FALSE;
   END_IF;
   #读UID指令 := #_w3 AND (#读UID定时器.ET >= T#300ms) AND NOT #IO状态1[3] AND NOT #IO状态2[3] AND NOT #IO状态4[3] AND NOT #IO状态3[3];
   IF #读UID指令 THEN #清除指令 := FALSE; END_IF;
   #_w4 := #配置完成定时器.Q AND NOT #IO状态1[3];
   #判断定时器_1.TON(IN := #_w4, PT := T#2S);   // TON coil
   #IO故障_1 := #_w4 AND #判断定时器_1.Q;
   IF #IO故障_1 THEN
       #IO输出值_1[0] := 16#39;
       #IO输出值_1[1] := 16#39;
       #IO输出值_1[2] := 16#39;
       #IO输出值_1[3] := 16#39;
       #IO输出值_1[4] := 16#39;
       #IO输出值_1[5] := 16#39;
   END_IF;
   #_w5 := #配置完成定时器.Q AND NOT #IO状态2[3];
   #判断定时器_2.TON(IN := #_w5, PT := T#2S);   // TON coil
   #IO故障_2 := #_w5 AND #判断定时器_2.Q;
   IF #IO故障_2 THEN
       #IO输出值_2[0] := 16#39;
       #IO输出值_2[1] := 16#39;
       #IO输出值_2[2] := 16#39;
       #IO输出值_2[3] := 16#39;
       #IO输出值_2[4] := 16#39;
       #IO输出值_2[5] := 16#39;
   END_IF;
   #_w6 := #配置完成定时器.Q AND NOT #IO状态3[3];
   #判断定时器_3.TON(IN := #_w6, PT := T#2S);   // TON coil
   #IO故障_3 := #_w6 AND #判断定时器_3.Q;
   IF #IO故障_3 THEN
       #IO输出值_3[0] := 16#39;
       #IO输出值_3[1] := 16#39;
       #IO输出值_3[2] := 16#39;
       #IO输出值_3[3] := 16#39;
       #IO输出值_3[4] := 16#39;
       #IO输出值_3[5] := 16#39;
   END_IF;
   #_w7 := #配置完成定时器.Q AND NOT #IO状态4[3];
   #判断定时器_4.TON(IN := #_w7, PT := T#2S);   // TON coil
   #IO故障_4 := #_w7 AND #判断定时器_4.Q;
   IF #IO故障_4 THEN
       #IO输出值_4[0] := 16#39;
       #IO输出值_4[1] := 16#39;
       #IO输出值_4[2] := 16#39;
       #IO输出值_4[3] := 16#39;
       #IO输出值_4[4] := 16#39;
       #IO输出值_4[5] := 16#39;
   END_IF;
   #_w8 := #读UID定时器.Q AND ((#IO状态1[0] AND (#栈板有无_1 <> 1)) OR (NOT #IO状态1[0] AND (#栈板有无_1 = 1))) AND #IO状态1[3] AND NOT #IO故障_1;
   #UID状态值_1 := #_w8 AND #读取过滤定时器_5.Q;
   #读取过滤定时器_5.TON(IN := #_w8, PT := T#2s);   // TON coil
   #_w9 := #读UID定时器.Q AND ((#IO状态2[0] AND (#栈板有无_2 <> 1)) OR (NOT #IO状态2[0] AND (#栈板有无_2 = 1))) AND #IO状态2[3] AND NOT #IO故障_2;
   #UID状态值_2 := #_w9 AND #读取过滤定时器_6.Q;
   #读取过滤定时器_6.TON(IN := #_w9, PT := T#2s);   // TON coil
   #_w10 := #读UID定时器.Q AND ((#IO状态3[0] AND (#栈板有无_3 <> 1)) OR (NOT #IO状态3[0] AND (#栈板有无_3 = 1))) AND #IO状态3[3] AND NOT #IO故障_3;
   #UID状态值_3 := #_w10 AND #读取过滤定时器_7.Q;
   #读取过滤定时器_7.TON(IN := #_w10, PT := T#2s);   // TON coil
   #_w11 := #读UID定时器.Q AND ((#IO状态4[0] AND (#栈板有无_4 <> 1)) OR (NOT #IO状态4[0] AND (#栈板有无_4 = 1))) AND #IO状态4[3] AND NOT #IO故障_4;
   #UID状态值_4 := #_w11 AND #读取过滤定时器_8.Q;
   #读取过滤定时器_8.TON(IN := #_w11, PT := T#2s);   // TON coil
   #_w12 := #UID状态值_1 OR #UID状态值_2 OR #UID状态值_3 OR #UID状态值_4 OR #中断连接 OR "FirstScan";
   #_w13 := #_w12 AND NOT #读取P;   // rising edge
   #读取P := #_w12;
   IF #_w13 AND #读取完成 THEN
       #IO成功_1 := FALSE;
       #IO成功_2 := FALSE;
       #IO成功_3 := FALSE;
       #IO成功_4 := FALSE;
       #IO故障_2 := FALSE;
       #IO故障_1 := FALSE;
       #IO故障_3 := FALSE;
       #IO故障_4 := FALSE;
       #次数1 := 0;
       #次数2 := 0;
       #次数3 := 0;
       #次数4 := 0;
   END_IF;
   #读取完成 := (#IO成功_1 OR #IO故障_2) AND (#IO成功_2 OR #IO故障_1) AND (#IO成功_3 OR #IO故障_3) AND (#IO成功_4 OR #IO故障_4);
END_REGION

REGION Network 2
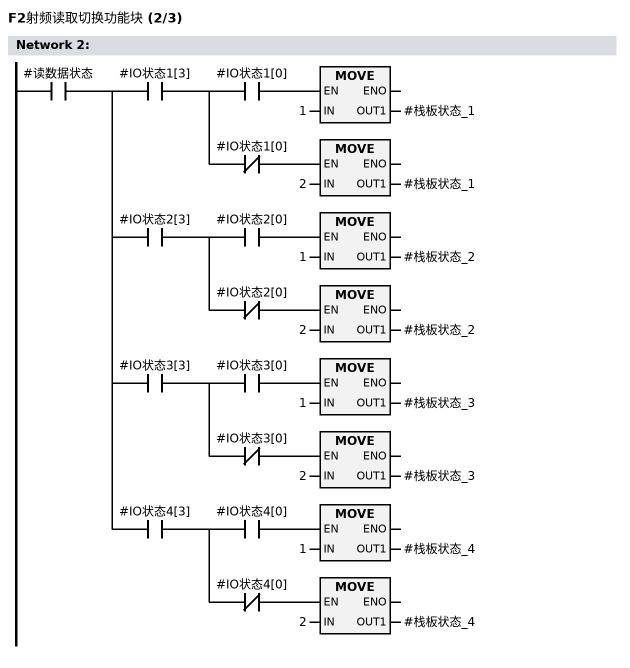
   RUNG wire#powerrail
      Contact( #读数据状态 )
      wire#w1
      Contact( #IO状态1[3] )
      wire#w2
      Contact( #IO状态1[0] )
      Move(in := 1, out1 => #栈板状态_1)
   END_RUNG
   RUNG wire#w2
      I_Contact( #IO状态1[0] )
      Move(in := 2, out1 => #栈板状态_1)
   END_RUNG
   RUNG wire#w1
      Contact( #IO状态2[3] )
      wire#w3
      Contact( #IO状态2[0] )
      Move(in := 1, out1 => #栈板状态_2)
   END_RUNG
   RUNG wire#w3
      I_Contact( #IO状态2[0] )
      Move(in := 2, out1 => #栈板状态_2)
   END_RUNG
   RUNG wire#w1
      Contact( #IO状态3[3] )
      wire#w4
      Contact( #IO状态3[0] )
      Move(in := 1, out1 => #栈板状态_3)
   END_RUNG
   RUNG wire#w4
      I_Contact( #IO状态3[0] )
      Move(in := 2, out1 => #栈板状态_3)
   END_RUNG
   RUNG wire#w1
      Contact( #IO状态4[3] )
      wire#w5
      Contact( #IO状态4[0] )
      Move(in := 1, out1 => #栈板状态_4)
   END_RUNG
   RUNG wire#w5
      I_Contact( #IO状态4[0] )
      Move(in := 2, out1 => #栈板状态_4)
   END_RUNG
   // the same network as SCL:
   #_w1 := #读数据状态 AND #IO状态1[3];
   IF #_w1 AND #IO状态1[0] THEN #栈板状态_1 := 1; END_IF;
   IF #_w1 AND NOT #IO状态1[0] THEN #栈板状态_1 := 2; END_IF;
   #_w2 := #读数据状态 AND #IO状态2[3];
   IF #_w2 AND #IO状态2[0] THEN #栈板状态_2 := 1; END_IF;
   IF #_w2 AND NOT #IO状态2[0] THEN #栈板状态_2 := 2; END_IF;
   #_w3 := #读数据状态 AND #IO状态3[3];
   IF #_w3 AND #IO状态3[0] THEN #栈板状态_3 := 1; END_IF;
   IF #_w3 AND NOT #IO状态3[0] THEN #栈板状态_3 := 2; END_IF;
   #_w4 := #读数据状态 AND #IO状态4[3];
   IF #_w4 AND #IO状态4[0] THEN #栈板状态_4 := 1; END_IF;
   IF #_w4 AND NOT #IO状态4[0] THEN #栈板状态_4 := 2; END_IF;
END_REGION

REGION Network 3
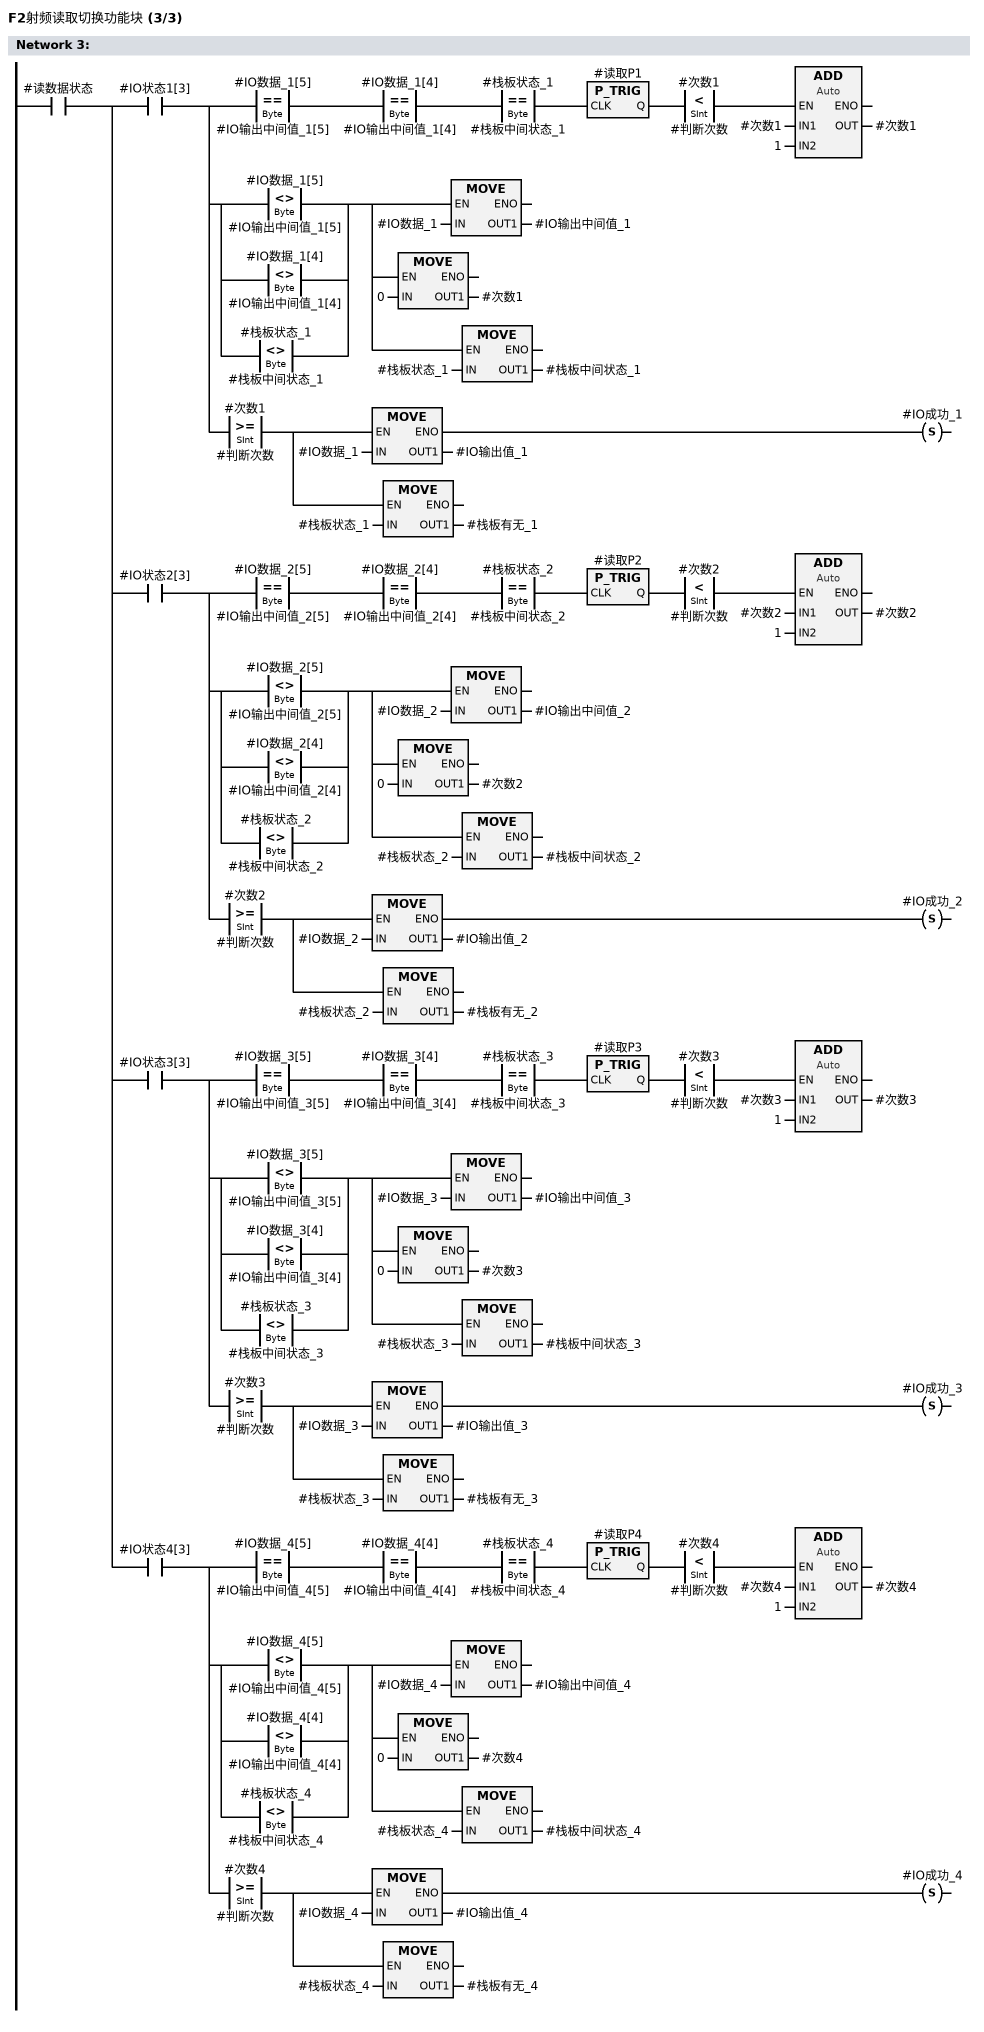
   RUNG wire#powerrail
      Contact( #读数据状态 )
      wire#w1
      Contact( #IO状态1[3] )
      wire#w2
      { S7_Templates := "SrcType := Byte" } EQ_Contact(in1 := #IO数据_1[5], in2 := #IO输出中间值_1[5])
      { S7_Templates := "SrcType := Byte" } EQ_Contact(in1 := #IO数据_1[4], in2 := #IO输出中间值_1[4])
      { S7_Templates := "SrcType := Byte" } EQ_Contact(in1 := #栈板状态_1, in2 := #栈板中间状态_1)
      P_Trig( #读取P1 )
      { S7_Templates := "SrcType := SInt" } LT_Contact(in1 := #次数1, in2 := #判断次数)
      Add(in1 := #次数1, in2 := 1, out => #次数1)
   END_RUNG
   RUNG wire#w2
      { S7_Templates := "SrcType := Byte" } NE_Contact(in1 := #IO数据_1[5], in2 := #IO输出中间值_1[5])
      wire#w3
      Move(in := #IO数据_1, out1 => #IO输出中间值_1)
   END_RUNG
   RUNG wire#w2
      { S7_Templates := "SrcType := Byte" } NE_Contact(in1 := #IO数据_1[4], in2 := #IO输出中间值_1[4])
   END_RUNG wire#w3
   RUNG wire#w2
      { S7_Templates := "SrcType := Byte" } NE_Contact(in1 := #栈板状态_1, in2 := #栈板中间状态_1)
   END_RUNG wire#w3
   RUNG wire#w3
      Move(in := 0, out1 => #次数1)
   END_RUNG
   RUNG wire#w3
      Move(in := #栈板状态_1, out1 => #栈板中间状态_1)
   END_RUNG
   RUNG wire#w2
      { S7_Templates := "SrcType := SInt" } GE_Contact(in1 := #次数1, in2 := #判断次数)
      wire#w4
      Move(in := #IO数据_1, out1 => #IO输出值_1)
      S_Coil( #IO成功_1 )
   END_RUNG
   RUNG wire#w4
      Move(in := #栈板状态_1, out1 => #栈板有无_1)
   END_RUNG
   RUNG wire#w1
      Contact( #IO状态2[3] )
      wire#w5
      { S7_Templates := "SrcType := Byte" } EQ_Contact(in1 := #IO数据_2[5], in2 := #IO输出中间值_2[5])
      { S7_Templates := "SrcType := Byte" } EQ_Contact(in1 := #IO数据_2[4], in2 := #IO输出中间值_2[4])
      { S7_Templates := "SrcType := Byte" } EQ_Contact(in1 := #栈板状态_2, in2 := #栈板中间状态_2)
      P_Trig( #读取P2 )
      { S7_Templates := "SrcType := SInt" } LT_Contact(in1 := #次数2, in2 := #判断次数)
      Add(in1 := #次数2, in2 := 1, out => #次数2)
   END_RUNG
   RUNG wire#w5
      { S7_Templates := "SrcType := Byte" } NE_Contact(in1 := #IO数据_2[5], in2 := #IO输出中间值_2[5])
      wire#w6
      Move(in := #IO数据_2, out1 => #IO输出中间值_2)
   END_RUNG
   RUNG wire#w5
      { S7_Templates := "SrcType := Byte" } NE_Contact(in1 := #IO数据_2[4], in2 := #IO输出中间值_2[4])
   END_RUNG wire#w6
   RUNG wire#w5
      { S7_Templates := "SrcType := Byte" } NE_Contact(in1 := #栈板状态_2, in2 := #栈板中间状态_2)
   END_RUNG wire#w6
   RUNG wire#w6
      Move(in := 0, out1 => #次数2)
   END_RUNG
   RUNG wire#w6
      Move(in := #栈板状态_2, out1 => #栈板中间状态_2)
   END_RUNG
   RUNG wire#w5
      { S7_Templates := "SrcType := SInt" } GE_Contact(in1 := #次数2, in2 := #判断次数)
      wire#w7
      Move(in := #IO数据_2, out1 => #IO输出值_2)
      S_Coil( #IO成功_2 )
   END_RUNG
   RUNG wire#w7
      Move(in := #栈板状态_2, out1 => #栈板有无_2)
   END_RUNG
   RUNG wire#w1
      Contact( #IO状态3[3] )
      wire#w8
      { S7_Templates := "SrcType := Byte" } EQ_Contact(in1 := #IO数据_3[5], in2 := #IO输出中间值_3[5])
      { S7_Templates := "SrcType := Byte" } EQ_Contact(in1 := #IO数据_3[4], in2 := #IO输出中间值_3[4])
      { S7_Templates := "SrcType := Byte" } EQ_Contact(in1 := #栈板状态_3, in2 := #栈板中间状态_3)
      P_Trig( #读取P3 )
      { S7_Templates := "SrcType := SInt" } LT_Contact(in1 := #次数3, in2 := #判断次数)
      Add(in1 := #次数3, in2 := 1, out => #次数3)
   END_RUNG
   RUNG wire#w8
      { S7_Templates := "SrcType := Byte" } NE_Contact(in1 := #IO数据_3[5], in2 := #IO输出中间值_3[5])
      wire#w9
      Move(in := #IO数据_3, out1 => #IO输出中间值_3)
   END_RUNG
   RUNG wire#w8
      { S7_Templates := "SrcType := Byte" } NE_Contact(in1 := #IO数据_3[4], in2 := #IO输出中间值_3[4])
   END_RUNG wire#w9
   RUNG wire#w8
      { S7_Templates := "SrcType := Byte" } NE_Contact(in1 := #栈板状态_3, in2 := #栈板中间状态_3)
   END_RUNG wire#w9
   RUNG wire#w9
      Move(in := 0, out1 => #次数3)
   END_RUNG
   RUNG wire#w9
      Move(in := #栈板状态_3, out1 => #栈板中间状态_3)
   END_RUNG
   RUNG wire#w8
      { S7_Templates := "SrcType := SInt" } GE_Contact(in1 := #次数3, in2 := #判断次数)
      wire#w10
      Move(in := #IO数据_3, out1 => #IO输出值_3)
      S_Coil( #IO成功_3 )
   END_RUNG
   RUNG wire#w10
      Move(in := #栈板状态_3, out1 => #栈板有无_3)
   END_RUNG
   RUNG wire#w1
      Contact( #IO状态4[3] )
      wire#w11
      { S7_Templates := "SrcType := Byte" } EQ_Contact(in1 := #IO数据_4[5], in2 := #IO输出中间值_4[5])
      { S7_Templates := "SrcType := Byte" } EQ_Contact(in1 := #IO数据_4[4], in2 := #IO输出中间值_4[4])
      { S7_Templates := "SrcType := Byte" } EQ_Contact(in1 := #栈板状态_4, in2 := #栈板中间状态_4)
      P_Trig( #读取P4 )
      { S7_Templates := "SrcType := SInt" } LT_Contact(in1 := #次数4, in2 := #判断次数)
      Add(in1 := #次数4, in2 := 1, out => #次数4)
   END_RUNG
   RUNG wire#w11
      { S7_Templates := "SrcType := Byte" } NE_Contact(in1 := #IO数据_4[5], in2 := #IO输出中间值_4[5])
      wire#w12
      Move(in := #IO数据_4, out1 => #IO输出中间值_4)
   END_RUNG
   RUNG wire#w11
      { S7_Templates := "SrcType := Byte" } NE_Contact(in1 := #IO数据_4[4], in2 := #IO输出中间值_4[4])
   END_RUNG wire#w12
   RUNG wire#w11
      { S7_Templates := "SrcType := Byte" } NE_Contact(in1 := #栈板状态_4, in2 := #栈板中间状态_4)
   END_RUNG wire#w12
   RUNG wire#w12
      Move(in := 0, out1 => #次数4)
   END_RUNG
   RUNG wire#w12
      Move(in := #栈板状态_4, out1 => #栈板中间状态_4)
   END_RUNG
   RUNG wire#w11
      { S7_Templates := "SrcType := SInt" } GE_Contact(in1 := #次数4, in2 := #判断次数)
      wire#w13
      Move(in := #IO数据_4, out1 => #IO输出值_4)
      S_Coil( #IO成功_4 )
   END_RUNG
   RUNG wire#w13
      Move(in := #栈板状态_4, out1 => #栈板有无_4)
   END_RUNG
   // the same network as SCL:
   #_w1 := #读数据状态 AND #IO状态1[3];
   #_w2 := #_w1 AND (#IO数据_1[5] = #IO输出中间值_1[5]) AND (#IO数据_1[4] = #IO输出中间值_1[4]) AND (#栈板状态_1 = #栈板中间状态_1);
   #_w3 := #_w2 AND NOT #读取P1;   // rising edge
   #读取P1 := #_w2;
   IF #_w3 AND (#次数1 < #判断次数) THEN #次数1 := #次数1 + 1; END_IF;
   #_w4 := #_w1 AND ((#IO数据_1[5] <> #IO输出中间值_1[5]) OR (#IO数据_1[4] <> #IO输出中间值_1[4]) OR (#栈板状态_1 <> #栈板中间状态_1));
   IF #_w4 THEN
       #IO输出中间值_1 := #IO数据_1;
       #次数1 := 0;
       #栈板中间状态_1 := #栈板状态_1;
   END_IF;
   IF #_w1 AND (#次数1 >= #判断次数) THEN
       #IO输出值_1 := #IO数据_1;
       #IO成功_1 := TRUE;
       #栈板有无_1 := #栈板状态_1;
   END_IF;
   #_w5 := #读数据状态 AND #IO状态2[3];
   #_w6 := #_w5 AND (#IO数据_2[5] = #IO输出中间值_2[5]) AND (#IO数据_2[4] = #IO输出中间值_2[4]) AND (#栈板状态_2 = #栈板中间状态_2);
   #_w7 := #_w6 AND NOT #读取P2;   // rising edge
   #读取P2 := #_w6;
   IF #_w7 AND (#次数2 < #判断次数) THEN #次数2 := #次数2 + 1; END_IF;
   #_w8 := #_w5 AND ((#IO数据_2[5] <> #IO输出中间值_2[5]) OR (#IO数据_2[4] <> #IO输出中间值_2[4]) OR (#栈板状态_2 <> #栈板中间状态_2));
   IF #_w8 THEN
       #IO输出中间值_2 := #IO数据_2;
       #次数2 := 0;
       #栈板中间状态_2 := #栈板状态_2;
   END_IF;
   IF #_w5 AND (#次数2 >= #判断次数) THEN
       #IO输出值_2 := #IO数据_2;
       #IO成功_2 := TRUE;
       #栈板有无_2 := #栈板状态_2;
   END_IF;
   #_w9 := #读数据状态 AND #IO状态3[3];
   #_w10 := #_w9 AND (#IO数据_3[5] = #IO输出中间值_3[5]) AND (#IO数据_3[4] = #IO输出中间值_3[4]) AND (#栈板状态_3 = #栈板中间状态_3);
   #_w11 := #_w10 AND NOT #读取P3;   // rising edge
   #读取P3 := #_w10;
   IF #_w11 AND (#次数3 < #判断次数) THEN #次数3 := #次数3 + 1; END_IF;
   #_w12 := #_w9 AND ((#IO数据_3[5] <> #IO输出中间值_3[5]) OR (#IO数据_3[4] <> #IO输出中间值_3[4]) OR (#栈板状态_3 <> #栈板中间状态_3));
   IF #_w12 THEN
       #IO输出中间值_3 := #IO数据_3;
       #次数3 := 0;
       #栈板中间状态_3 := #栈板状态_3;
   END_IF;
   IF #_w9 AND (#次数3 >= #判断次数) THEN
       #IO输出值_3 := #IO数据_3;
       #IO成功_3 := TRUE;
       #栈板有无_3 := #栈板状态_3;
   END_IF;
   #_w13 := #读数据状态 AND #IO状态4[3];
   #_w14 := #_w13 AND (#IO数据_4[5] = #IO输出中间值_4[5]) AND (#IO数据_4[4] = #IO输出中间值_4[4]) AND (#栈板状态_4 = #栈板中间状态_4);
   #_w15 := #_w14 AND NOT #读取P4;   // rising edge
   #读取P4 := #_w14;
   IF #_w15 AND (#次数4 < #判断次数) THEN #次数4 := #次数4 + 1; END_IF;
   #_w16 := #_w13 AND ((#IO数据_4[5] <> #IO输出中间值_4[5]) OR (#IO数据_4[4] <> #IO输出中间值_4[4]) OR (#栈板状态_4 <> #栈板中间状态_4));
   IF #_w16 THEN
       #IO输出中间值_4 := #IO数据_4;
       #次数4 := 0;
       #栈板中间状态_4 := #栈板状态_4;
   END_IF;
   IF #_w13 AND (#次数4 >= #判断次数) THEN
       #IO输出值_4 := #IO数据_4;
       #IO成功_4 := TRUE;
       #栈板有无_4 := #栈板状态_4;
   END_IF;
END_REGION
END_FUNCTION_BLOCK

FUNCTION "射频通信" : Void   // FC3, LAD
{ S7_Optimized_Access := 'TRUE' }
VERSION : 0.1
BEGIN

REGION Network 2: SP******************** 192 168 0 79
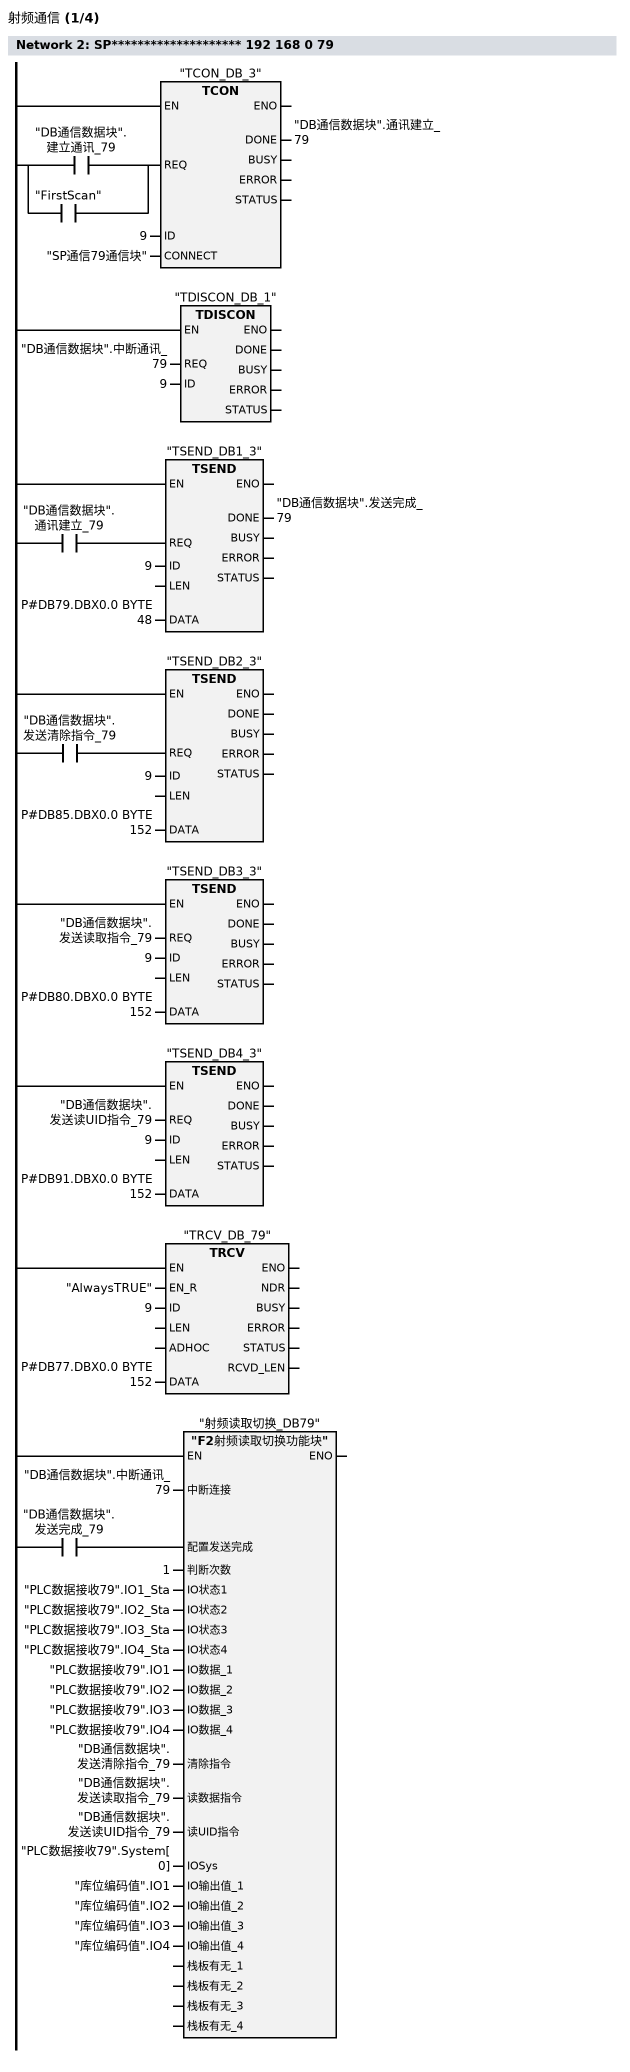
   "TCON_DB_3"(REQ := "DB通信数据块".建立通讯_79 OR "FirstScan",   // TCON
               ID := 9,
               CONNECT := "SP通信79通信块",
               DONE => "DB通信数据块".通讯建立_79);
   "TDISCON_DB_1"(REQ := "DB通信数据块".中断通讯_79, ID := 9);   // TDISCON
   "TSEND_DB1_3"(REQ := "DB通信数据块".通讯建立_79, ID := 9, DATA := P#DB79.DBX0.0 BYTE 48, DONE => "DB通信数据块".发送完成_79);   // TSEND
   "TSEND_DB2_3"(REQ := "DB通信数据块".发送清除指令_79, ID := 9, DATA := P#DB85.DBX0.0 BYTE 152);   // TSEND
   "TSEND_DB3_3"(REQ := "DB通信数据块".发送读取指令_79, ID := 9, DATA := P#DB80.DBX0.0 BYTE 152);   // TSEND
   "TSEND_DB4_3"(REQ := "DB通信数据块".发送读UID指令_79, ID := 9, DATA := P#DB91.DBX0.0 BYTE 152);   // TSEND
   "TRCV_DB_79"(EN_R := "AlwaysTRUE", ID := 9, DATA := P#DB77.DBX0.0 BYTE 152);   // TRCV
   "射频读取切换_DB79"(中断连接 := "DB通信数据块".中断通讯_79,   // "F2射频读取切换功能块"
                 配置发送完成 := "DB通信数据块".发送完成_79,
                 判断次数 := 1,
                 IO状态1 := "PLC数据接收79".IO1_Sta,
                 IO状态2 := "PLC数据接收79".IO2_Sta,
                 IO状态3 := "PLC数据接收79".IO3_Sta,
                 IO状态4 := "PLC数据接收79".IO4_Sta,
                 IO数据_1 := "PLC数据接收79".IO1,
                 IO数据_2 := "PLC数据接收79".IO2,
                 IO数据_3 := "PLC数据接收79".IO3,
                 IO数据_4 := "PLC数据接收79".IO4,
                 清除指令 := "DB通信数据块".发送清除指令_79,
                 读数据指令 := "DB通信数据块".发送读取指令_79,
                 读UID指令 := "DB通信数据块".发送读UID指令_79,
                 IOSys := "PLC数据接收79".System[0],
                 IO输出值_1 := "库位编码值".IO1,
                 IO输出值_2 := "库位编码值".IO2,
                 IO输出值_3 := "库位编码值".IO3,
                 IO输出值_4 := "库位编码值".IO4);
END_REGION

REGION Network 3: SP******************** 192 168 0 80
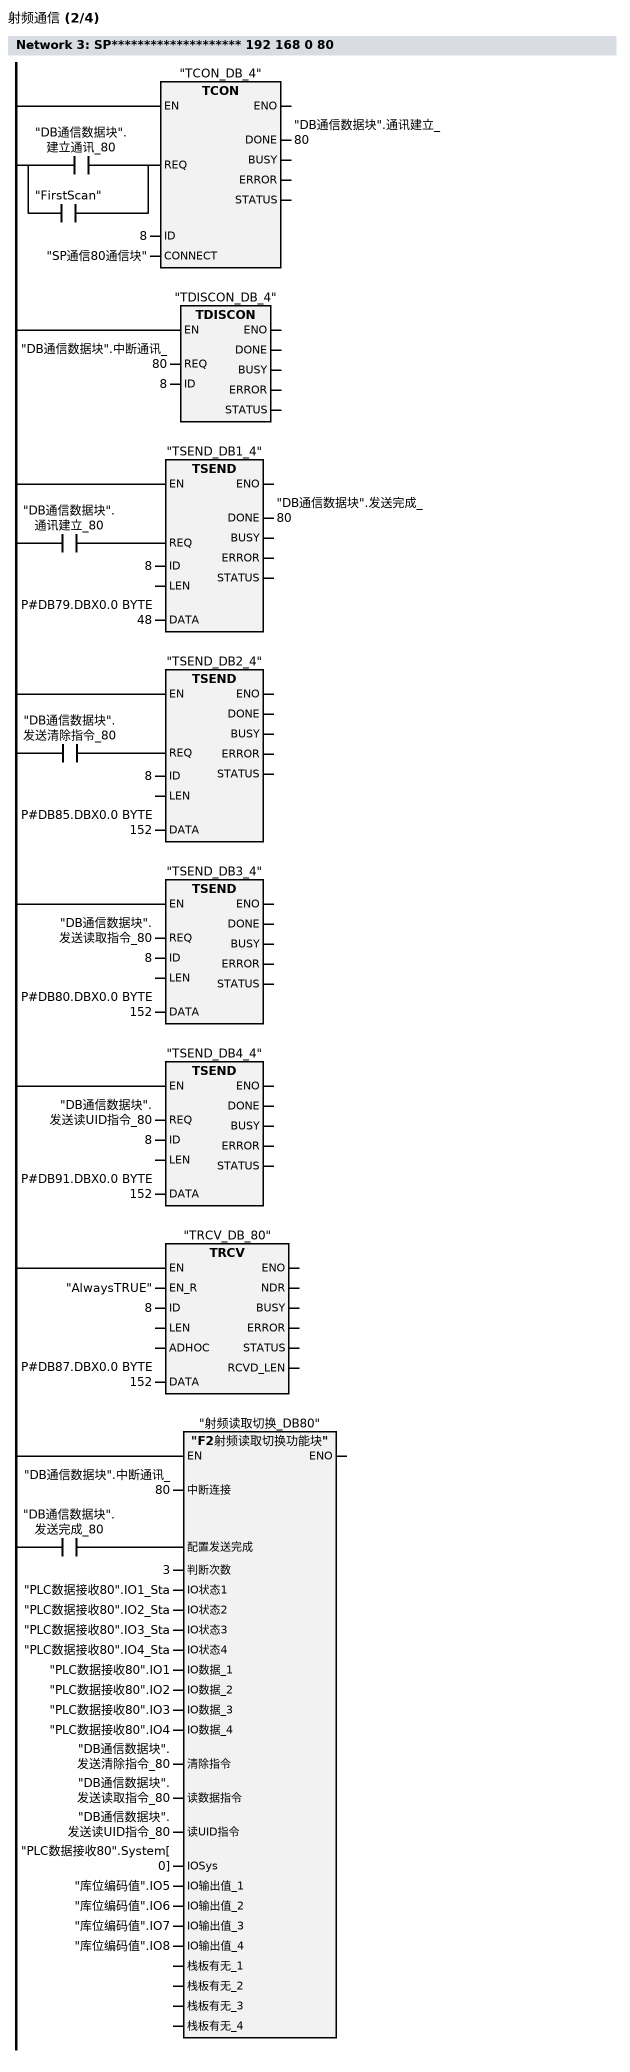
   "TCON_DB_4"(REQ := "DB通信数据块".建立通讯_80 OR "FirstScan",   // TCON
               ID := 8,
               CONNECT := "SP通信80通信块",
               DONE => "DB通信数据块".通讯建立_80);
   "TDISCON_DB_4"(REQ := "DB通信数据块".中断通讯_80, ID := 8);   // TDISCON
   "TSEND_DB1_4"(REQ := "DB通信数据块".通讯建立_80, ID := 8, DATA := P#DB79.DBX0.0 BYTE 48, DONE => "DB通信数据块".发送完成_80);   // TSEND
   "TSEND_DB2_4"(REQ := "DB通信数据块".发送清除指令_80, ID := 8, DATA := P#DB85.DBX0.0 BYTE 152);   // TSEND
   "TSEND_DB3_4"(REQ := "DB通信数据块".发送读取指令_80, ID := 8, DATA := P#DB80.DBX0.0 BYTE 152);   // TSEND
   "TSEND_DB4_4"(REQ := "DB通信数据块".发送读UID指令_80, ID := 8, DATA := P#DB91.DBX0.0 BYTE 152);   // TSEND
   "TRCV_DB_80"(EN_R := "AlwaysTRUE", ID := 8, DATA := P#DB87.DBX0.0 BYTE 152);   // TRCV
   "射频读取切换_DB80"(中断连接 := "DB通信数据块".中断通讯_80,   // "F2射频读取切换功能块"
                 配置发送完成 := "DB通信数据块".发送完成_80,
                 判断次数 := 3,
                 IO状态1 := "PLC数据接收80".IO1_Sta,
                 IO状态2 := "PLC数据接收80".IO2_Sta,
                 IO状态3 := "PLC数据接收80".IO3_Sta,
                 IO状态4 := "PLC数据接收80".IO4_Sta,
                 IO数据_1 := "PLC数据接收80".IO1,
                 IO数据_2 := "PLC数据接收80".IO2,
                 IO数据_3 := "PLC数据接收80".IO3,
                 IO数据_4 := "PLC数据接收80".IO4,
                 清除指令 := "DB通信数据块".发送清除指令_80,
                 读数据指令 := "DB通信数据块".发送读取指令_80,
                 读UID指令 := "DB通信数据块".发送读UID指令_80,
                 IOSys := "PLC数据接收80".System[0],
                 IO输出值_1 := "库位编码值".IO5,
                 IO输出值_2 := "库位编码值".IO6,
                 IO输出值_3 := "库位编码值".IO7,
                 IO输出值_4 := "库位编码值".IO8);
END_REGION

REGION Network 4: SP******************** 192 168 0 81
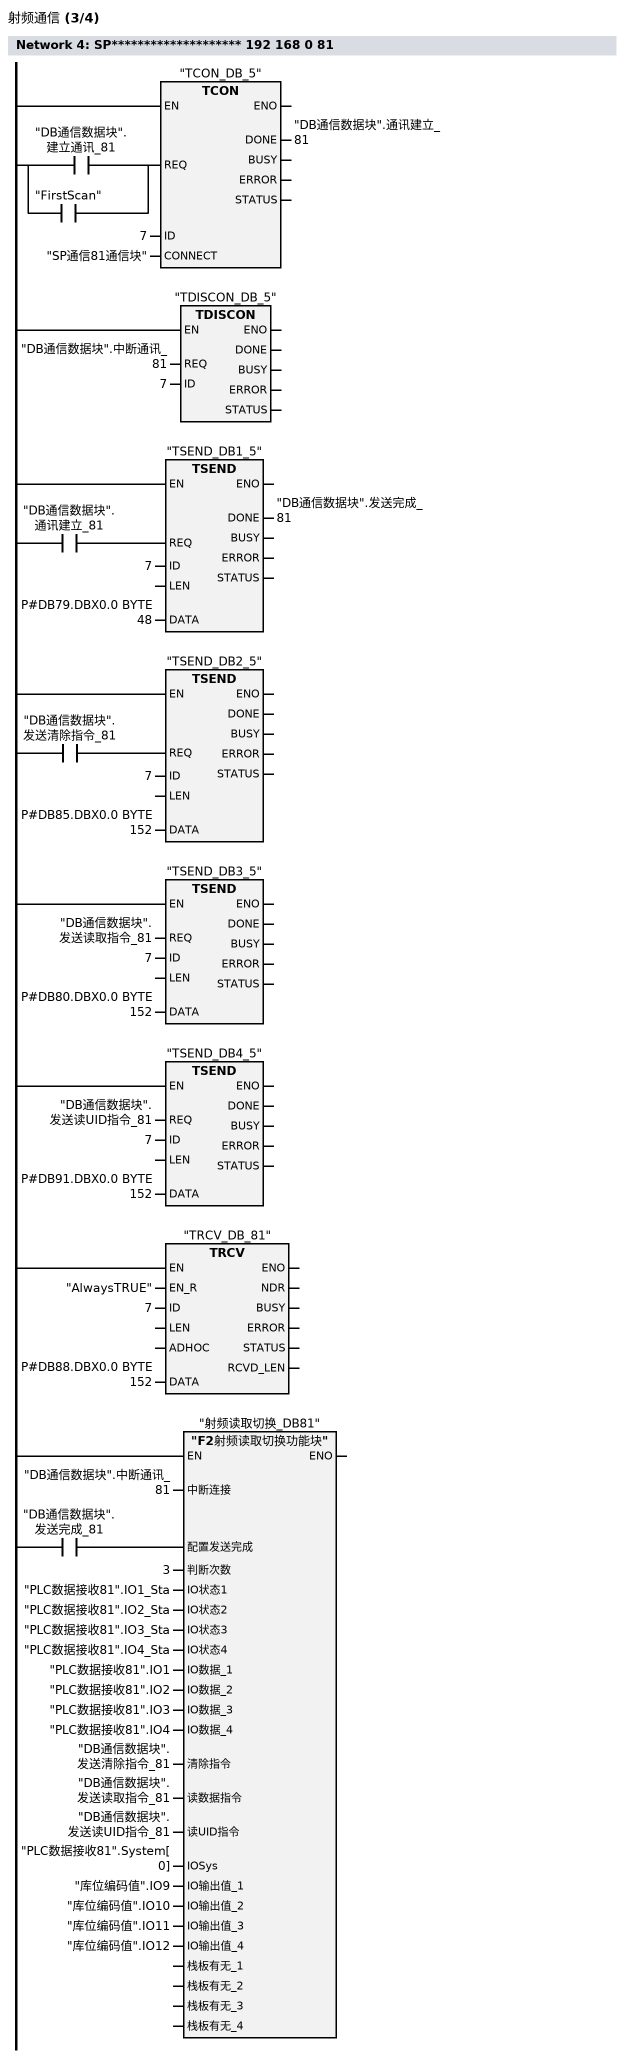
   "TCON_DB_5"(REQ := "DB通信数据块".建立通讯_81 OR "FirstScan",   // TCON
               ID := 7,
               CONNECT := "SP通信81通信块",
               DONE => "DB通信数据块".通讯建立_81);
   "TDISCON_DB_5"(REQ := "DB通信数据块".中断通讯_81, ID := 7);   // TDISCON
   "TSEND_DB1_5"(REQ := "DB通信数据块".通讯建立_81, ID := 7, DATA := P#DB79.DBX0.0 BYTE 48, DONE => "DB通信数据块".发送完成_81);   // TSEND
   "TSEND_DB2_5"(REQ := "DB通信数据块".发送清除指令_81, ID := 7, DATA := P#DB85.DBX0.0 BYTE 152);   // TSEND
   "TSEND_DB3_5"(REQ := "DB通信数据块".发送读取指令_81, ID := 7, DATA := P#DB80.DBX0.0 BYTE 152);   // TSEND
   "TSEND_DB4_5"(REQ := "DB通信数据块".发送读UID指令_81, ID := 7, DATA := P#DB91.DBX0.0 BYTE 152);   // TSEND
   "TRCV_DB_81"(EN_R := "AlwaysTRUE", ID := 7, DATA := P#DB88.DBX0.0 BYTE 152);   // TRCV
   "射频读取切换_DB81"(中断连接 := "DB通信数据块".中断通讯_81,   // "F2射频读取切换功能块"
                 配置发送完成 := "DB通信数据块".发送完成_81,
                 判断次数 := 3,
                 IO状态1 := "PLC数据接收81".IO1_Sta,
                 IO状态2 := "PLC数据接收81".IO2_Sta,
                 IO状态3 := "PLC数据接收81".IO3_Sta,
                 IO状态4 := "PLC数据接收81".IO4_Sta,
                 IO数据_1 := "PLC数据接收81".IO1,
                 IO数据_2 := "PLC数据接收81".IO2,
                 IO数据_3 := "PLC数据接收81".IO3,
                 IO数据_4 := "PLC数据接收81".IO4,
                 清除指令 := "DB通信数据块".发送清除指令_81,
                 读数据指令 := "DB通信数据块".发送读取指令_81,
                 读UID指令 := "DB通信数据块".发送读UID指令_81,
                 IOSys := "PLC数据接收81".System[0],
                 IO输出值_1 := "库位编码值".IO9,
                 IO输出值_2 := "库位编码值".IO10,
                 IO输出值_3 := "库位编码值".IO11,
                 IO输出值_4 := "库位编码值".IO12);
END_REGION

REGION Network 5: SP******************** 192 168 0 82
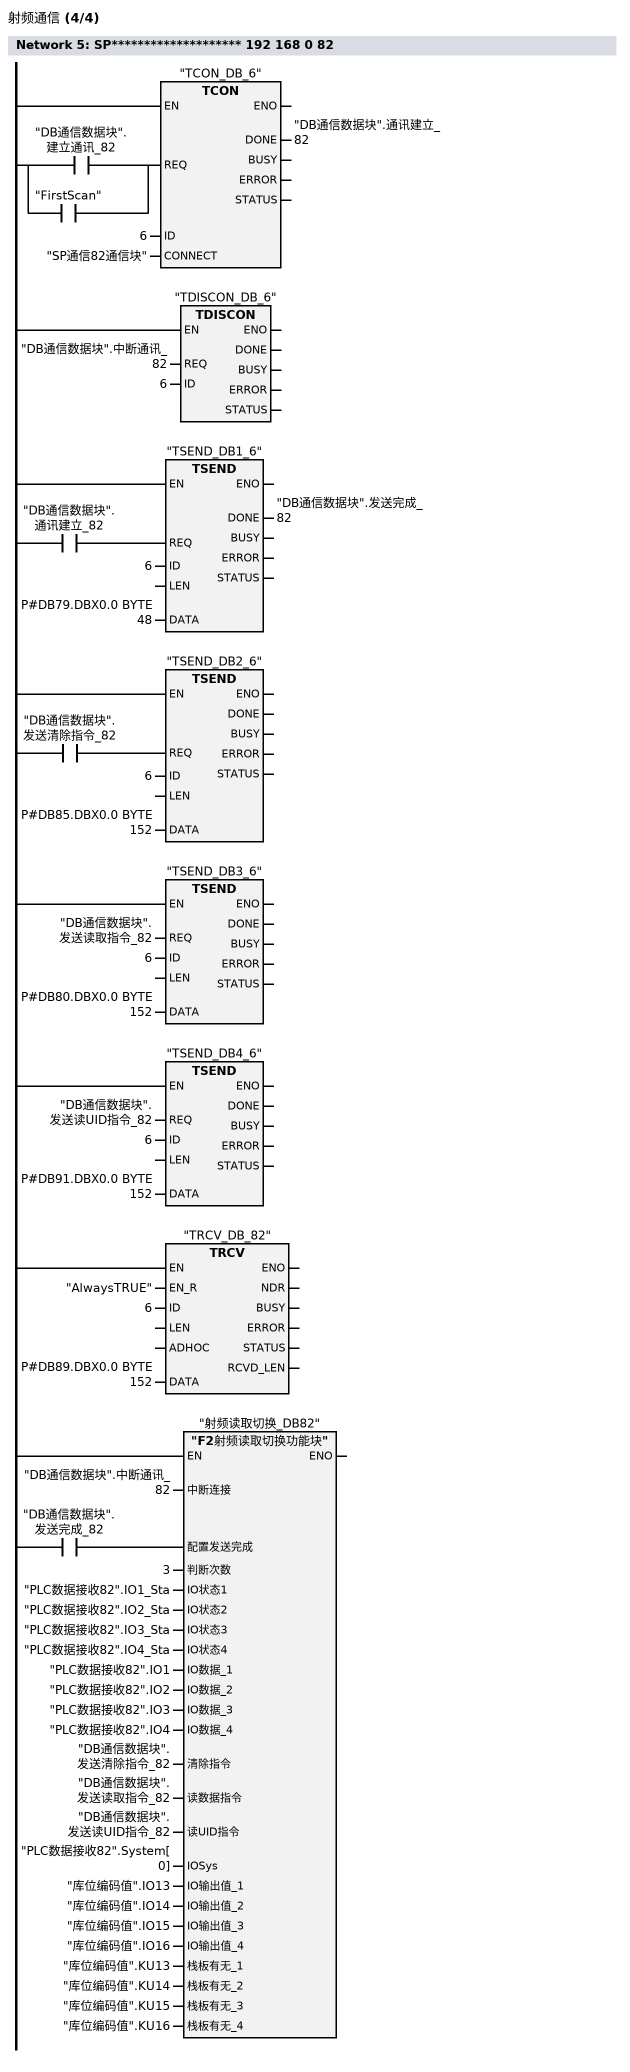
   "TCON_DB_6"(REQ := "DB通信数据块".建立通讯_82 OR "FirstScan",   // TCON
               ID := 6,
               CONNECT := "SP通信82通信块",
               DONE => "DB通信数据块".通讯建立_82);
   "TDISCON_DB_6"(REQ := "DB通信数据块".中断通讯_82, ID := 6);   // TDISCON
   "TSEND_DB1_6"(REQ := "DB通信数据块".通讯建立_82, ID := 6, DATA := P#DB79.DBX0.0 BYTE 48, DONE => "DB通信数据块".发送完成_82);   // TSEND
   "TSEND_DB2_6"(REQ := "DB通信数据块".发送清除指令_82, ID := 6, DATA := P#DB85.DBX0.0 BYTE 152);   // TSEND
   "TSEND_DB3_6"(REQ := "DB通信数据块".发送读取指令_82, ID := 6, DATA := P#DB80.DBX0.0 BYTE 152);   // TSEND
   "TSEND_DB4_6"(REQ := "DB通信数据块".发送读UID指令_82, ID := 6, DATA := P#DB91.DBX0.0 BYTE 152);   // TSEND
   "TRCV_DB_82"(EN_R := "AlwaysTRUE", ID := 6, DATA := P#DB89.DBX0.0 BYTE 152);   // TRCV
   "射频读取切换_DB82"(中断连接 := "DB通信数据块".中断通讯_82,   // "F2射频读取切换功能块"
                 配置发送完成 := "DB通信数据块".发送完成_82,
                 判断次数 := 3,
                 IO状态1 := "PLC数据接收82".IO1_Sta,
                 IO状态2 := "PLC数据接收82".IO2_Sta,
                 IO状态3 := "PLC数据接收82".IO3_Sta,
                 IO状态4 := "PLC数据接收82".IO4_Sta,
                 IO数据_1 := "PLC数据接收82".IO1,
                 IO数据_2 := "PLC数据接收82".IO2,
                 IO数据_3 := "PLC数据接收82".IO3,
                 IO数据_4 := "PLC数据接收82".IO4,
                 清除指令 := "DB通信数据块".发送清除指令_82,
                 读数据指令 := "DB通信数据块".发送读取指令_82,
                 读UID指令 := "DB通信数据块".发送读UID指令_82,
                 IOSys := "PLC数据接收82".System[0],
                 IO输出值_1 := "库位编码值".IO13,
                 IO输出值_2 := "库位编码值".IO14,
                 IO输出值_3 := "库位编码值".IO15,
                 IO输出值_4 := "库位编码值".IO16,
                 栈板有无_1 := "库位编码值".KU13,
                 栈板有无_2 := "库位编码值".KU14,
                 栈板有无_3 := "库位编码值".KU15,
                 栈板有无_4 := "库位编码值".KU16);
END_REGION
END_FUNCTION